KUKA KRL program: EPS_2_25694_AR02_A_20260223033033.src

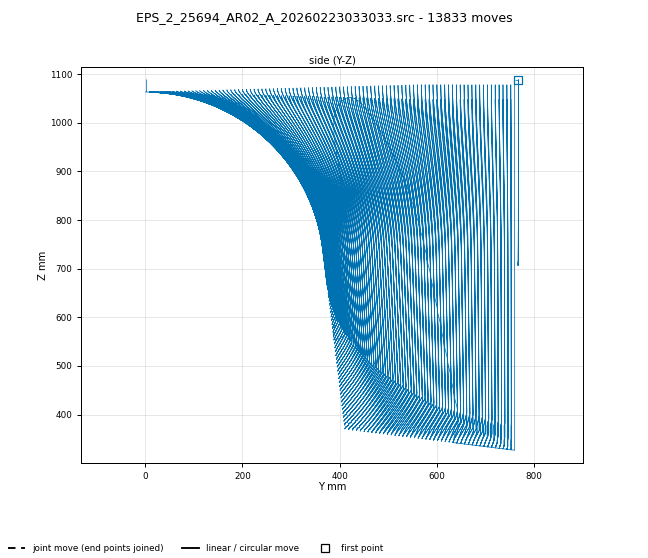
[picture p0: tool path of EPS_2_25694_AR02_A_20260223033033.src, 13833 of 13835 moves have a stored position in this frame; points joined in program order, loops and branches not executed]
&ACCESS RVP
&REL 4
&COMMENT QRS 19112012
&PARAM EDITMASK = *
DEF PART()
EXT BAS (BAS_COMMAND :IN,REAL :IN )
INT I
BAS (#INITMOV,0 )

;KUKA QRS Post kuka4.cps  Date:22-06-2017 !

File_ID=3049

QRS_PRE_INIT()

;Init var - Until changes are made in qrs_pre_init
Outlet_Square_prg=0
Inlet_1_Square_prg=0
Inlet_2_Square_prg=0
Inlet_3_Square_prg=0
Inlet_4_Square_prg=0
Inlet_5_Square_prg=0

Outlet_1={X 0.000, Y 562.000, Z 735.500, B 0.000, E1 0.000 }
Inlet_1={X 0.000, Y 562.000, Z 705.500, B 0.000, E1 180.000 }
Outlet_1_type=686
Inlet_1_type=686
;QRS#1=Sidecore dimensions
;QRS#2=675-27" Concrete
;QRS#3=675-27" Concrete
;QRS#4=
;QRS#5=
;QRS#6=
;QRS#7=
;QRS#8=
;QRS#9=S306-38L
;QRS#10=S306-38L
;QRS#11=
;QRS#12=
;QRS#13=
;QRS#14=
;QRS#15=
;QRS#16=1524x152x1524 5'
;QRS#17=EPS Height
;QRS#18=1078,5
;QRS#19=*
;QRS#20= UPDATED VERSION 22-06-2017
;QRS#21=*
Outlet_Square=0550
Inlet_1_Square=0550
Inlet_2_Square=0
Inlet_3_Square=0
Inlet_4_Square=0
Inlet_5_Square=0
Mill_Square=1
Outlet_Square_Prg=265
Inlet_1_Square_prg=265

QRS_INIT()

$ADVANCE=5

; T1
PTP {E1 173.041,E2 173.041}
PTP {X 0,Y 767.71,A -85,B 0,C 180,E1 173.041,E2 173.041,E3 0,E4 0,E5 0,E6 0}
QRS_SPEED_INIT()
LIN {X 0,Y 767.71,Z 1088.5,A -85,B 0,C 180,E1 173.041,E2 173.041,E3 0,E4 0,E5 0,E6 0} C_VEL
LIN {X 0,Y 767.71,Z 709.31,A -85,B 0,C 180,E1 173.041,E2 173.041} C_VEL
LIN {X 0,Y 767.737,Z 707.31,A -85,B 0,C 180,E1 173.19,E2 173.19} C_VEL
LIN {X 0,Y 767.796,Z 707.31,A -85,B 0,C 180,E1 173.458,E2 173.458} C_VEL
LIN {X 0,Y 767.812,Z 707.31,A -85,B 0,C 180,E1 177.201,E2 177.201} C_VEL
LIN {X 0,Y 767.839,Z 707.31,A -85,B 0,C 180,E1 180.933,E2 180.933} C_VEL
LIN {X 0,Y 767.833,Z 707.31,A -85,B 0,C 180,E1 184.668,E2 184.668} C_VEL
LIN {X 0,Y 767.857,Z 707.31,A -85,B 0,C 180,E1 188.423,E2 188.423} C_VEL
LIN {X 0,Y 767.829,Z 707.31,A -85,B 0,C 180,E1 192.215,E2 192.215} C_VEL
LIN {X 0,Y 767.83,Z 707.31,A -85,B 0,C 180,E1 196.204,E2 196.204} C_VEL
LIN {X 0,Y 767.77,Z 707.31,A -85,B 0,C 180,E1 199.988,E2 199.988} C_VEL
LIN {X 0,Y 767.749,Z 707.31,A -85,B 0,C 180,E1 204.013,E2 204.013} C_VEL
LIN {X 0,Y 767.75,Z 707.31,A -85,B 0,C 180,E1 208.167,E2 208.167} C_VEL
LIN {X 0,Y 767.324,Z 707.31,A -85,B 0,C 180,E1 210.324,E2 210.324} C_VEL
LIN {X 0,Y 767.754,Z 707.31,A -85,B 0,C 180,E1 212.49,E2 212.49} C_VEL
LIN {X 0,Y 767.43,Z 707.31,A -85,B 0,C 180,E1 213.85,E2 213.85} C_VEL
LIN {X 0,Y 767.706,Z 707.31,A -85,B 0,C 180,E1 217.094,E2 217.094} C_VEL
LIN {X 0,Y 767.088,Z 707.31,A -85,B 0,C 180,E1 220.03,E2 220.03} C_VEL
LIN {X 0,Y 767.533,Z 707.31,A -85,B 0,C 180,E1 221.88,E2 221.88} C_VEL
LIN {X 0,Y 767.581,Z 707.31,A -85,B 0,C 180,E1 222.891,E2 222.891} C_VEL
LIN {X 0,Y 767.581,Z 707.31,A -85,B 0,C 180,E1 227.109,E2 227.109} C_VEL
LIN {X 0,Y 767.53,Z 707.31,A -85,B 0,C 180,E1 228.12,E2 228.12} C_VEL
LIN {X 0,Y 767.102,Z 707.31,A -85,B 0,C 180,E1 230.553,E2 230.553} C_VEL
LIN {X 0,Y 767.692,Z 707.31,A -85,B 0,C 180,E1 232.964,E2 232.964} C_VEL
LIN {X 0,Y 767.598,Z 707.31,A -85,B 0,C 180,E1 236.132,E2 236.132} C_VEL
LIN {X 0,Y 767.614,Z 707.31,A -85,B 0,C 180,E1 237.503,E2 237.503} C_VEL
LIN {X 0,Y 767.641,Z 707.31,A -85,B 0,C 180,E1 239.69,E2 239.69} C_VEL
LIN {X 0,Y 767.411,Z 728.971,A -85,B 0,C 180,E1 240.873,E2 240.873} C_VEL
LIN {X 0,Y 767.537,Z 761.793,A -85,B 0,C 180,E1 241.233,E2 241.233} C_VEL
LIN {X 0,Y 767.433,Z 775.286,A -85,B 0,C 180,E1 241.406,E2 241.406} C_VEL
LIN {X 0,Y 767.548,Z 791.123,A -85,B 0,C 180,E1 241.677,E2 241.677} C_VEL
LIN {X 0,Y 767.449,Z 807.75,A -85,B 0,C 180,E1 242.019,E2 242.019} C_VEL
LIN {X 0,Y 767.663,Z 824.864,A -85,B 0,C 180,E1 242.456,E2 242.456} C_VEL
LIN {X 0,Y 767.66,Z 840.823,A -85,B 0,C 180,E1 242.921,E2 242.921} C_VEL
LIN {X 0,Y 767.553,Z 854.893,A -85,B 0,C 180,E1 243.38,E2 243.38} C_VEL
LIN {X 0,Y 767.694,Z 871.263,A -85,B 0,C 180,E1 243.998,E2 243.998} C_VEL
LIN {X 0,Y 767.655,Z 888.029,A -85,B 0,C 180,E1 244.706,E2 244.706} C_VEL
LIN {X 0,Y 767.705,Z 901.802,A -85,B 0,C 180,E1 245.351,E2 245.351} C_VEL
LIN {X 0,Y 767.712,Z 916.578,A -85,B 0,C 180,E1 246.114,E2 246.114} C_VEL
LIN {X 0,Y 767.693,Z 930.073,A -85,B 0,C 180,E1 246.876,E2 246.876} C_VEL
LIN {X 0,Y 767.691,Z 942.43,A -85,B 0,C 180,E1 247.634,E2 247.634} C_VEL
LIN {X 0,Y 767.701,Z 955.671,A -85,B 0,C 180,E1 248.523,E2 248.523} C_VEL
LIN {X 0,Y 767.718,Z 968.193,A -85,B 0,C 180,E1 249.439,E2 249.439} C_VEL
LIN {X 0,Y 767.619,Z 980.057,A -85,B 0,C 180,E1 250.38,E2 250.38} C_VEL
LIN {X 0,Y 767.656,Z 990.133,A -85,B 0,C 180,E1 251.245,E2 251.245} C_VEL
LIN {X 0,Y 767.778,Z 1000.684,A -85,B 0,C 180,E1 252.23,E2 252.23} C_VEL
LIN {X 0,Y 767.637,Z 1011.458,A -85,B 0,C 180,E1 253.326,E2 253.326} C_VEL
LIN {X 0,Y 767.699,Z 1020.42,A -85,B 0,C 180,E1 254.322,E2 254.322} C_VEL
LIN {X 0,Y 767.767,Z 1028.417,A -85,B 0,C 180,E1 255.29,E2 255.29} C_VEL
LIN {X 0,Y 767.624,Z 1037.823,A -85,B 0,C 180,E1 256.546,E2 256.546} C_VEL
LIN {X 0,Y 767.75,Z 1044.548,A -85,B 0,C 180,E1 257.545,E2 257.545} C_VEL
LIN {X 0,Y 767.749,Z 1048.907,A -85,B 0,C 180,E1 258.26,E2 258.26} C_VEL
LIN {X 0,Y 767.595,Z 1053.115,A -85,B 0,C 180,E1 258.971,E2 258.971} C_VEL
LIN {X 0,Y 767.579,Z 1059.347,A -85,B 0,C 180,E1 260.157,E2 260.157} C_VEL
LIN {X 0,Y 767.814,Z 1064.751,A -85,B 0,C 180,E1 261.341,E2 261.341} C_VEL
LIN {X 0,Y 767.552,Z 1069.482,A -85,B 0,C 180,E1 262.516,E2 262.516} C_VEL
LIN {X 0,Y 767.638,Z 1073.816,A -85,B 0,C 180,E1 263.832,E2 263.832} C_VEL
LIN {X 0,Y 767.832,Z 1075.821,A -85,B 0,C 180,E1 264.583,E2 264.583} C_VEL
LIN {X 0,Y 767.656,Z 1077.679,A -85,B 0,C 180,E1 265.331,E2 265.331} C_VEL
LIN {X 0,Y 767.552,Z 1079.276,A -85,B 0,C 180,E1 266.079,E2 266.079} C_VEL
LIN {X 0,Y 767.665,Z 1081.027,A -85,B 0,C 180,E1 267.201,E2 267.201} C_VEL
LIN {X 0,Y 767.713,Z 1082.196,A -85,B 0,C 180,E1 268.321,E2 268.321} C_VEL
LIN {X 0,Y 767.556,Z 1082.708,A -85,B 0,C 180,E1 269.067,E2 269.067} C_VEL
LIN {X 0,Y 767.7,Z 1082.68,A -85,B 0,C 180,E1 270.933,E2 270.933} C_VEL
LIN {X 0,Y 767.651,Z 1081.876,A -85,B 0,C 180,E1 272.052,E2 272.052} C_VEL
LIN {X 0,Y 767.525,Z 1081.053,A -85,B 0,C 180,E1 272.8,E2 272.8} C_VEL
LIN {X 0,Y 767.569,Z 1079.273,A -85,B 0,C 180,E1 273.921,E2 273.921} C_VEL
LIN {X 0,Y 767.76,Z 1077.66,A -85,B 0,C 180,E1 274.668,E2 274.668} C_VEL
LIN {X 0,Y 767.653,Z 1074.831,A -85,B 0,C 180,E1 275.793,E2 275.793} C_VEL
LIN {X 0,Y 767.602,Z 1072.628,A -85,B 0,C 180,E1 276.544,E2 276.544} C_VEL
LIN {X 0,Y 767.713,Z 1069.455,A -85,B 0,C 180,E1 277.483,E2 277.483} C_VEL
LIN {X 0,Y 767.824,Z 1067.577,A -85,B 0,C 180,E1 277.952,E2 277.952} C_VEL
LIN {X 0,Y 767.62,Z 1063.757,A -85,B 0,C 180,E1 278.897,E2 278.897} C_VEL
LIN {X 0,Y 767.559,Z 1058.195,A -85,B 0,C 180,E1 280.08,E2 280.08} C_VEL
LIN {X 0,Y 767.835,Z 1051.779,A -85,B 0,C 180,E1 281.263,E2 281.263} C_VEL
LIN {X 0,Y 767.624,Z 1044.562,A -85,B 0,C 180,E1 282.457,E2 282.457} C_VEL
LIN {X 0,Y 767.658,Z 1036.703,A -85,B 0,C 180,E1 283.612,E2 283.612} C_VEL
LIN {X 0,Y 767.821,Z 1029.879,A -85,B 0,C 180,E1 284.516,E2 284.516} C_VEL
LIN {X 0,Y 767.629,Z 1020.425,A -85,B 0,C 180,E1 285.679,E2 285.679} C_VEL
LIN {X 0,Y 767.731,Z 1009.176,A -85,B 0,C 180,E1 286.916,E2 286.916} C_VEL
LIN {X 0,Y 767.752,Z 999.435,A -85,B 0,C 180,E1 287.893,E2 287.893} C_VEL
LIN {X 0,Y 767.658,Z 988.765,A -85,B 0,C 180,E1 288.878,E2 288.878} C_VEL
LIN {X 0,Y 767.742,Z 977.061,A -85,B 0,C 180,E1 289.864,E2 289.864} C_VEL
LIN {X 0,Y 767.717,Z 964.937,A -85,B 0,C 180,E1 290.806,E2 290.806} C_VEL
LIN {X 0,Y 767.695,Z 954,A -85,B 0,C 180,E1 291.594,E2 291.594} C_VEL
LIN {X 0,Y 767.712,Z 940.408,A -85,B 0,C 180,E1 292.491,E2 292.491} C_VEL
LIN {X 0,Y 767.708,Z 926.801,A -85,B 0,C 180,E1 293.314,E2 293.314} C_VEL
LIN {X 0,Y 767.702,Z 913.126,A -85,B 0,C 180,E1 294.071,E2 294.071} C_VEL
LIN {X 0,Y 767.609,Z 898.313,A -85,B 0,C 180,E1 294.82,E2 294.82} C_VEL
LIN {X 0,Y 767.699,Z 884.655,A -85,B 0,C 180,E1 295.444,E2 295.444} C_VEL
LIN {X 0,Y 767.675,Z 869.453,A -85,B 0,C 180,E1 296.074,E2 296.074} C_VEL
LIN {X 0,Y 767.622,Z 855.717,A -85,B 0,C 180,E1 296.587,E2 296.587} C_VEL
LIN {X 0,Y 767.679,Z 837.479,A -85,B 0,C 180,E1 297.183,E2 297.183} C_VEL
LIN {X 0,Y 767.517,Z 820.548,A -85,B 0,C 180,E1 297.665,E2 297.665} C_VEL
LIN {X 0,Y 767.57,Z 810.447,A -85,B 0,C 180,E1 297.91,E2 297.91} C_VEL
LIN {X 0,Y 767.621,Z 801.598,A -85,B 0,C 180,E1 298.106,E2 298.106} C_VEL
LIN {X 0,Y 767.599,Z 787.941,A -85,B 0,C 180,E1 298.38,E2 298.38} C_VEL
LIN {X 0,Y 767.429,Z 775.322,A -85,B 0,C 180,E1 298.593,E2 298.593} C_VEL
LIN {X 0,Y 767.549,Z 757.094,A -85,B 0,C 180,E1 298.825,E2 298.825} C_VEL
LIN {X 0,Y 767.411,Z 729.395,A -85,B 0,C 180,E1 299.122,E2 299.122} C_VEL
LIN {X 0,Y 767.689,Z 707.31,A -85,B 0,C 180,E1 300.308,E2 300.308} C_VEL
LIN {X 0,Y 767.796,Z 707.31,A -85,B 0,C 180,E1 302.488,E2 302.488} C_VEL
LIN {X 0,Y 767.259,Z 707.31,A -85,B 0,C 180,E1 304.756,E2 304.756} C_VEL
LIN {X 0,Y 767.698,Z 707.31,A -85,B 0,C 180,E1 307.093,E2 307.093} C_VEL
LIN {X 0,Y 767.134,Z 707.31,A -85,B 0,C 180,E1 310.034,E2 310.034} C_VEL
LIN {X 0,Y 767.63,Z 707.31,A -85,B 0,C 180,E1 311.873,E2 311.873} C_VEL
LIN {X 0,Y 767.669,Z 707.31,A -85,B 0,C 180,E1 312.898,E2 312.898} C_VEL
LIN {X 0,Y 767.67,Z 707.31,A -85,B 0,C 180,E1 314.427,E2 314.427} C_VEL
LIN {X 0,Y 767.632,Z 707.31,A -85,B 0,C 180,E1 315.57,E2 315.57} C_VEL
LIN {X 0,Y 767.641,Z 707.31,A -85,B 0,C 180,E1 319.92,E2 319.92} C_VEL
LIN {X 0,Y 767.641,Z 707.31,A -85,B 0,C 180,E1 320.586,E2 320.586} C_VEL
LIN {X 0,Y 767.199,Z 707.31,A -85,B 0,C 180,E1 322.956,E2 322.956} C_VEL
LIN {X 0,Y 767.714,Z 707.31,A -85,B 0,C 180,E1 325.268,E2 325.268} C_VEL
LIN {X 0,Y 767.766,Z 707.31,A -85,B 0,C 180,E1 329.62,E2 329.62} C_VEL
LIN {X 0,Y 767.768,Z 707.31,A -85,B 0,C 180,E1 333.539,E2 333.539} C_VEL
LIN {X 0,Y 767.758,Z 707.31,A -85,B 0,C 180,E1 333.929,E2 333.929} C_VEL
LIN {X 0,Y 767.757,Z 707.31,A -85,B 0,C 180,E1 338.014,E2 338.014} C_VEL
LIN {X 0,Y 767.788,Z 707.31,A -85,B 0,C 180,E1 341.985,E2 341.985} C_VEL
LIN {X 0,Y 767.515,Z 707.31,A -85,B 0,C 180,E1 343.931,E2 343.931} C_VEL
LIN {X 0,Y 767.673,Z 707.31,A -85,B 0,C 180,E1 345.866,E2 345.866} C_VEL
LIN {X 0,Y 767.85,Z 707.31,A -85,B 0,C 180,E1 349.687,E2 349.687} C_VEL
LIN {X 0,Y 767.871,Z 707.31,A -85,B 0,C 180,E1 353.458,E2 353.458} C_VEL
LIN {X 0,Y 767.844,Z 707.31,A -85,B 0,C 180,E1 357.201,E2 357.201} C_VEL
LIN {X 0,Y 767.813,Z 707.31,A -85,B 0,C 180,E1 360.933,E2 360.933} C_VEL
LIN {X 0,Y 767.806,Z 707.31,A -85,B 0,C 180,E1 364.668,E2 364.668} C_VEL
LIN {X 0,Y 767.794,Z 707.31,A -85,B 0,C 180,E1 368.424,E2 368.424} C_VEL
LIN {X 0,Y 767.808,Z 707.31,A -85,B 0,C 180,E1 372.216,E2 372.216} C_VEL
LIN {X 0,Y 767.849,Z 707.31,A -85,B 0,C 180,E1 376.209,E2 376.209} C_VEL
LIN {X 0,Y 767.798,Z 707.31,A -85,B 0,C 180,E1 379.987,E2 379.987} C_VEL
LIN {X 0,Y 767.788,Z 707.31,A -85,B 0,C 180,E1 384.011,E2 384.011} C_VEL
LIN {X 0,Y 767.772,Z 707.31,A -85,B 0,C 180,E1 388.166,E2 388.166} C_VEL
LIN {X 0,Y 767.323,Z 707.31,A -85,B 0,C 180,E1 390.324,E2 390.324} C_VEL
LIN {X 0,Y 767.706,Z 707.31,A -85,B 0,C 180,E1 392.493,E2 392.493} C_VEL
LIN {X 0,Y 767.384,Z 707.31,A -85,B 0,C 180,E1 393.845,E2 393.845} C_VEL
LIN {X 0,Y 767.666,Z 707.31,A -85,B 0,C 180,E1 397.09,E2 397.09} C_VEL
LIN {X 0,Y 767.085,Z 707.31,A -85,B 0,C 180,E1 400.03,E2 400.03} C_VEL
LIN {X 0,Y 767.568,Z 707.31,A -85,B 0,C 180,E1 401.877,E2 401.877} C_VEL
LIN {X 0,Y 767.619,Z 707.31,A -85,B 0,C 180,E1 402.894,E2 402.894} C_VEL
LIN {X 0,Y 767.576,Z 707.31,A -85,B 0,C 180,E1 407.109,E2 407.109} C_VEL
LIN {X 0,Y 767.531,Z 707.31,A -85,B 0,C 180,E1 408.12,E2 408.12} C_VEL
LIN {X 0,Y 767.121,Z 707.31,A -85,B 0,C 180,E1 410.555,E2 410.555} C_VEL
LIN {X 0,Y 767.734,Z 707.31,A -85,B 0,C 180,E1 412.967,E2 412.967} C_VEL
LIN {X 0,Y 767.634,Z 707.31,A -85,B 0,C 180,E1 416.127,E2 416.127} C_VEL
LIN {X 0,Y 767.601,Z 707.31,A -85,B 0,C 180,E1 417.503,E2 417.503} C_VEL
LIN {X 0,Y 767.858,Z 707.31,A -85,B 0,C 180,E1 420.635,E2 420.635} C_VEL
LIN {X 0,Y 766.716,Z 707.31,A -85,B 0,C 180,E1 420.886,E2 420.886} C_VEL
LIN {X 0,Y 767.333,Z 731.466,A -85,B 0,C 180,E1 421.176,E2 421.176} C_VEL
LIN {X 0,Y 767.435,Z 745.357,A -85,B 0,C 180,E1 421.363,E2 421.363} C_VEL
LIN {X 0,Y 767.54,Z 761.823,A -85,B 0,C 180,E1 421.646,E2 421.646} C_VEL
LIN {X 0,Y 767.454,Z 778.242,A -85,B 0,C 180,E1 421.986,E2 421.986} C_VEL
LIN {X 0,Y 767.631,Z 794.143,A -85,B 0,C 180,E1 422.389,E2 422.389} C_VEL
LIN {X 0,Y 767.586,Z 811.017,A -85,B 0,C 180,E1 422.879,E2 422.879} C_VEL
LIN {X 0,Y 767.597,Z 821.633,A -85,B 0,C 180,E1 423.229,E2 423.229} C_VEL
LIN {X 0,Y 767.652,Z 830.77,A -85,B 0,C 180,E1 423.557,E2 423.557} C_VEL
LIN {X 0,Y 767.67,Z 842.534,A -85,B 0,C 180,E1 424.005,E2 424.005} C_VEL
LIN {X 0,Y 767.616,Z 857.298,A -85,B 0,C 180,E1 424.625,E2 424.625} C_VEL
LIN {X 0,Y 767.704,Z 872.822,A -85,B 0,C 180,E1 425.358,E2 425.358} C_VEL
LIN {X 0,Y 767.706,Z 886.246,A -85,B 0,C 180,E1 426.05,E2 426.05} C_VEL
LIN {X 0,Y 767.699,Z 900.808,A -85,B 0,C 180,E1 426.876,E2 426.876} C_VEL
LIN {X 0,Y 767.715,Z 913.106,A -85,B 0,C 180,E1 427.635,E2 427.635} C_VEL
LIN {X 0,Y 767.732,Z 926.109,A -85,B 0,C 180,E1 428.51,E2 428.51} C_VEL
LIN {X 0,Y 767.692,Z 937.694,A -85,B 0,C 180,E1 429.354,E2 429.354} C_VEL
LIN {X 0,Y 767.693,Z 949.134,A -85,B 0,C 180,E1 430.258,E2 430.258} C_VEL
LIN {X 0,Y 767.755,Z 960.62,A -85,B 0,C 180,E1 431.248,E2 431.248} C_VEL
LIN {X 0,Y 767.617,Z 971.133,A -85,B 0,C 180,E1 432.226,E2 432.226} C_VEL
LIN {X 0,Y 767.635,Z 980.763,A -85,B 0,C 180,E1 433.204,E2 433.204} C_VEL
LIN {X 0,Y 767.794,Z 990.787,A -85,B 0,C 180,E1 434.324,E2 434.324} C_VEL
LIN {X 0,Y 767.595,Z 998.788,A -85,B 0,C 180,E1 435.287,E2 435.287} C_VEL
LIN {X 0,Y 767.635,Z 1008.181,A -85,B 0,C 180,E1 436.555,E2 436.555} C_VEL
LIN {X 0,Y 767.838,Z 1014.839,A -85,B 0,C 180,E1 437.546,E2 437.546} C_VEL
LIN {X 0,Y 767.606,Z 1022.075,A -85,B 0,C 180,E1 438.734,E2 438.734} C_VEL
LIN {X 0,Y 767.688,Z 1028.418,A -85,B 0,C 180,E1 439.922,E2 439.922} C_VEL
LIN {X 0,Y 767.815,Z 1031.726,A -85,B 0,C 180,E1 440.633,E2 440.633} C_VEL
LIN {X 0,Y 767.696,Z 1033.956,A -85,B 0,C 180,E1 441.104,E2 441.104} C_VEL
LIN {X 0,Y 767.567,Z 1039.63,A -85,B 0,C 180,E1 442.516,E2 442.516} C_VEL
LIN {X 0,Y 767.836,Z 1043.902,A -85,B 0,C 180,E1 443.833,E2 443.833} C_VEL
LIN {X 0,Y 767.651,Z 1045.978,A -85,B 0,C 180,E1 444.582,E2 444.582} C_VEL
LIN {X 0,Y 767.527,Z 1047.797,A -85,B 0,C 180,E1 445.33,E2 445.33} C_VEL
LIN {X 0,Y 767.528,Z 1049.376,A -85,B 0,C 180,E1 446.079,E2 446.079} C_VEL
LIN {X 0,Y 767.766,Z 1051.076,A -85,B 0,C 180,E1 447.201,E2 447.201} C_VEL
LIN {X 0,Y 767.683,Z 1051.909,A -85,B 0,C 180,E1 447.948,E2 447.948} C_VEL
LIN {X 0,Y 767.503,Z 1052.73,A -85,B 0,C 180,E1 449.067,E2 449.067} C_VEL
LIN {X 0,Y 767.839,Z 1052.64,A -85,B 0,C 180,E1 450.933,E2 450.933} C_VEL
LIN {X 0,Y 767.651,Z 1052.167,A -85,B 0,C 180,E1 451.679,E2 451.679} C_VEL
LIN {X 0,Y 767.568,Z 1050.977,A -85,B 0,C 180,E1 452.8,E2 452.8} C_VEL
LIN {X 0,Y 767.769,Z 1049.14,A -85,B 0,C 180,E1 453.92,E2 453.92} C_VEL
LIN {X 0,Y 767.722,Z 1047.573,A -85,B 0,C 180,E1 454.669,E2 454.669} C_VEL
LIN {X 0,Y 767.556,Z 1044.725,A -85,B 0,C 180,E1 455.794,E2 455.794} C_VEL
LIN {X 0,Y 767.553,Z 1043.709,A -85,B 0,C 180,E1 456.169,E2 456.169} C_VEL
LIN {X 0,Y 767.803,Z 1039.283,A -85,B 0,C 180,E1 457.482,E2 457.482} C_VEL
LIN {X 0,Y 767.581,Z 1033.551,A -85,B 0,C 180,E1 458.898,E2 458.898} C_VEL
LIN {X 0,Y 767.696,Z 1027.934,A -85,B 0,C 180,E1 460.078,E2 460.078} C_VEL
LIN {X 0,Y 767.795,Z 1024.114,A -85,B 0,C 180,E1 460.788,E2 460.788} C_VEL
LIN {X 0,Y 767.632,Z 1020.089,A -85,B 0,C 180,E1 461.504,E2 461.504} C_VEL
LIN {X 0,Y 767.584,Z 1014.26,A -85,B 0,C 180,E1 462.458,E2 462.458} C_VEL
LIN {X 0,Y 767.802,Z 1006.2,A -85,B 0,C 180,E1 463.63,E2 463.63} C_VEL
LIN {X 0,Y 767.611,Z 998.056,A -85,B 0,C 180,E1 464.713,E2 464.713} C_VEL
LIN {X 0,Y 767.603,Z 988.335,A -85,B 0,C 180,E1 465.874,E2 465.874} C_VEL
LIN {X 0,Y 767.79,Z 978.725,A -85,B 0,C 180,E1 466.915,E2 466.915} C_VEL
LIN {X 0,Y 767.663,Z 968.946,A -85,B 0,C 180,E1 467.895,E2 467.895} C_VEL
LIN {X 0,Y 767.674,Z 958.234,A -85,B 0,C 180,E1 468.878,E2 468.878} C_VEL
LIN {X 0,Y 767.733,Z 946.486,A -85,B 0,C 180,E1 469.865,E2 469.865} C_VEL
LIN {X 0,Y 767.676,Z 936.03,A -85,B 0,C 180,E1 470.683,E2 470.683} C_VEL
LIN {X 0,Y 767.702,Z 923.158,A -85,B 0,C 180,E1 471.605,E2 471.605} C_VEL
LIN {X 0,Y 767.72,Z 909.669,A -85,B 0,C 180,E1 472.491,E2 472.491} C_VEL
LIN {X 0,Y 767.698,Z 897.13,A -85,B 0,C 180,E1 473.251,E2 473.251} C_VEL
LIN {X 0,Y 767.661,Z 883.363,A -85,B 0,C 180,E1 474.016,E2 474.016} C_VEL
LIN {X 0,Y 767.709,Z 868.143,A -85,B 0,C 180,E1 474.779,E2 474.779} C_VEL
LIN {X 0,Y 767.676,Z 854.017,A -85,B 0,C 180,E1 475.427,E2 475.427} C_VEL
LIN {X 0,Y 767.64,Z 840.173,A -85,B 0,C 180,E1 476.003,E2 476.003} C_VEL
LIN {X 0,Y 767.674,Z 822.353,A -85,B 0,C 180,E1 476.655,E2 476.655} C_VEL
LIN {X 0,Y 767.539,Z 807.048,A -85,B 0,C 180,E1 477.155,E2 477.155} C_VEL
LIN {X 0,Y 767.67,Z 790.049,A -85,B 0,C 180,E1 477.626,E2 477.626} C_VEL
LIN {X 0,Y 767.643,Z 774.248,A -85,B 0,C 180,E1 478.006,E2 478.006} C_VEL
LIN {X 0,Y 767.488,Z 760.439,A -85,B 0,C 180,E1 478.294,E2 478.294} C_VEL
LIN {X 0,Y 767.647,Z 741.352,A -85,B 0,C 180,E1 478.599,E2 478.599} C_VEL
LIN {X 0,Y 767.413,Z 720.586,A -85,B 0,C 180,E1 478.855,E2 478.855} C_VEL
LIN {X 0,Y 767.103,Z 715.733,A -85,B 0,C 180,E1 478.919,E2 478.919} C_VEL
LIN {X 0,Y 765.967,Z 707.31,A -85,B 0,C 180,E1 479.059,E2 479.059} C_VEL
LIN {X 0,Y 767.879,Z 707.31,A -85,B 0,C 180,E1 479.317,E2 479.317} C_VEL
LIN {X 0,Y 767.752,Z 707.31,A -85,B 0,C 180,E1 482.49,E2 482.49} C_VEL
LIN {X 0,Y 767.418,Z 707.31,A -85,B 0,C 180,E1 483.848,E2 483.848} C_VEL
LIN {X 0,Y 767.742,Z 707.31,A -85,B 0,C 180,E1 487.098,E2 487.098} C_VEL
LIN {X 0,Y 767.157,Z 707.31,A -85,B 0,C 180,E1 490.036,E2 490.036} C_VEL
LIN {X 0,Y 767.638,Z 707.31,A -85,B 0,C 180,E1 491.873,E2 491.873} C_VEL
LIN {X 0,Y 767.66,Z 707.31,A -85,B 0,C 180,E1 492.897,E2 492.897} C_VEL
LIN {X 0,Y 767.674,Z 707.31,A -85,B 0,C 180,E1 494.427,E2 494.427} C_VEL
LIN {X 0,Y 767.645,Z 707.31,A -85,B 0,C 180,E1 495.571,E2 495.571} C_VEL
LIN {X 0,Y 767.662,Z 707.31,A -85,B 0,C 180,E1 499.919,E2 499.919} C_VEL
LIN {X 0,Y 767.649,Z 707.31,A -85,B 0,C 180,E1 500.587,E2 500.587} C_VEL
LIN {X 0,Y 767.201,Z 707.31,A -85,B 0,C 180,E1 502.956,E2 502.956} C_VEL
LIN {X 0,Y 767.688,Z 707.31,A -85,B 0,C 180,E1 505.267,E2 505.267} C_VEL
LIN {X 0,Y 767.773,Z 707.31,A -85,B 0,C 180,E1 509.619,E2 509.619} C_VEL
LIN {X 0,Y 767.792,Z 707.31,A -85,B 0,C 180,E1 513.536,E2 513.536} C_VEL
LIN {X 0,Y 767.79,Z 707.31,A -85,B 0,C 180,E1 513.93,E2 513.93} C_VEL
LIN {X 0,Y 767.81,Z 707.31,A -85,B 0,C 180,E1 518.016,E2 518.016} C_VEL
LIN {X 0,Y 767.831,Z 707.31,A -85,B 0,C 180,E1 521.987,E2 521.987} C_VEL
LIN {X 0,Y 767.502,Z 707.31,A -85,B 0,C 180,E1 523.93,E2 523.93} C_VEL
LIN {X 0,Y 767.619,Z 707.31,A -85,B 0,C 180,E1 525.865,E2 525.865} C_VEL
LIN {X 0,Y 767.814,Z 707.31,A -85,B 0,C 180,E1 529.686,E2 529.686} C_VEL
LIN {X 0,Y 767.737,Z 707.31,A -85,B 0,C 180,E1 533.19,E2 533.19} C_VEL
LIN {X 0,Y 767.797,Z 709.31,A -85,B 0,C 180,E1 533.34,E2 533.34} C_VEL
LIN {X 0,Y 767.797,Z 1088.5,A -85,B 0,C 180,E1 533.34,E2 533.34} C_VEL
LIN {X 0,Y 767.797,Z 1088.5,A -85,B 0,C 180,E1 533.34,E2 533.34}

QRS_NEXT_CUT()
PTP {E1 537.316,E2 537.316}
PTP {X 0,Y 759.845,A -85,B 0,C 180,E1 537.316,E2 537.316,E3 0,E4 0,E5 0,E6 0}
QRS_SPEED_INIT()
LIN {X 0,Y 759.845,Z 1088.5,A -85,B 0,C 180,E1 537.316,E2 537.316,E3 0,E4 0,E5 0,E6 0} C_VEL
LIN {X 0,Y 759.845,Z 336.65,A -85,B 0,C 180,E1 537.316,E2 537.316} C_VEL
LIN {X 0,Y 759.845,Z 328.572,A -85,B 0,C 180,E1 537.316,E2 537.316} C_VEL
LIN {X 0,Y 759.845,Z 326.572,A -85,B 0,C 180,E1 537.165,E2 537.165} C_VEL
LIN {X 0,Y 759.903,Z 326.568,A -85,B 0,C 180,E1 534.488,E2 534.488} C_VEL
LIN {X 0,Y 759.869,Z 326.575,A -85,B 0,C 180,E1 531.601,E2 531.601} C_VEL
LIN {X 0,Y 759.845,Z 326.572,A -85,B 0,C 180,E1 529.077,E2 529.077} C_VEL
LIN {X 0,Y 759.89,Z 326.569,A -85,B 0,C 180,E1 526.454,E2 526.454} C_VEL
LIN {X 0,Y 759.873,Z 326.575,A -85,B 0,C 180,E1 523.487,E2 523.487} C_VEL
LIN {X 0,Y 759.846,Z 326.572,A -85,B 0,C 180,E1 520.953,E2 520.953} C_VEL
LIN {X 0,Y 759.881,Z 326.569,A -85,B 0,C 180,E1 518.381,E2 518.381} C_VEL
LIN {X 0,Y 759.873,Z 326.575,A -85,B 0,C 180,E1 515.346,E2 515.346} C_VEL
LIN {X 0,Y 759.847,Z 326.572,A -85,B 0,C 180,E1 512.817,E2 512.817} C_VEL
LIN {X 0,Y 759.891,Z 326.568,A -85,B 0,C 180,E1 510.173,E2 510.173} C_VEL
LIN {X 0,Y 759.87,Z 326.575,A -85,B 0,C 180,E1 507.17,E2 507.17} C_VEL
LIN {X 0,Y 759.848,Z 326.572,A -85,B 0,C 180,E1 504.62,E2 504.62} C_VEL
LIN {X 0,Y 759.899,Z 326.568,A -85,B 0,C 180,E1 501.989,E2 501.989} C_VEL
LIN {X 0,Y 759.873,Z 326.575,A -85,B 0,C 180,E1 499.052,E2 499.052} C_VEL
LIN {X 0,Y 759.849,Z 326.572,A -85,B 0,C 180,E1 496.474,E2 496.474} C_VEL
LIN {X 0,Y 759.916,Z 326.567,A -85,B 0,C 180,E1 493.749,E2 493.749} C_VEL
LIN {X 0,Y 759.866,Z 326.575,A -85,B 0,C 180,E1 490.832,E2 490.832} C_VEL
LIN {X 0,Y 759.85,Z 326.572,A -85,B 0,C 180,E1 488.301,E2 488.301} C_VEL
LIN {X 0,Y 759.911,Z 326.569,A -85,B 0,C 180,E1 485.593,E2 485.593} C_VEL
LIN {X 0,Y 759.85,Z 326.665,A -85,B 0,C 180,E1 484.249,E2 484.249} C_VEL
LIN {X 0,Y 759.884,Z 347.573,A -85,B 0,C 180,E1 482.756,E2 482.756} C_VEL
LIN {X 0,Y 759.914,Z 586.155,A -85,B 0,C 180,E1 480.163,E2 480.163} C_VEL
LIN {X 0,Y 759.918,Z 735.836,A -85,B 0,C 180,E1 478.552,E2 478.552} C_VEL
LIN {X 0,Y 759.897,Z 759.154,A -85,B 0,C 180,E1 478.189,E2 478.189} C_VEL
LIN {X 0,Y 759.902,Z 781.501,A -85,B 0,C 180,E1 477.701,E2 477.701} C_VEL
LIN {X 0,Y 759.897,Z 801.388,A -85,B 0,C 180,E1 477.167,E2 477.167} C_VEL
LIN {X 0,Y 759.919,Z 824.793,A -85,B 0,C 180,E1 476.406,E2 476.406} C_VEL
LIN {X 0,Y 759.916,Z 845.178,A -85,B 0,C 180,E1 475.61,E2 475.61} C_VEL
LIN {X 0,Y 759.913,Z 864.717,A -85,B 0,C 180,E1 474.735,E2 474.735} C_VEL
LIN {X 0,Y 759.912,Z 886.993,A -85,B 0,C 180,E1 473.578,E2 473.578} C_VEL
LIN {X 0,Y 759.914,Z 904.978,A -85,B 0,C 180,E1 472.513,E2 472.513} C_VEL
LIN {X 0,Y 759.906,Z 925.463,A -85,B 0,C 180,E1 471.133,E2 471.133} C_VEL
LIN {X 0,Y 759.916,Z 942.7,A -85,B 0,C 180,E1 469.815,E2 469.815} C_VEL
LIN {X 0,Y 759.916,Z 959.761,A -85,B 0,C 180,E1 468.329,E2 468.329} C_VEL
LIN {X 0,Y 759.898,Z 975.058,A -85,B 0,C 180,E1 466.827,E2 466.827} C_VEL
LIN {X 0,Y 759.912,Z 989.594,A -85,B 0,C 180,E1 465.179,E2 465.179} C_VEL
LIN {X 0,Y 759.908,Z 1001.089,A -85,B 0,C 180,E1 463.7,E2 463.7} C_VEL
LIN {X 0,Y 759.903,Z 1012.978,A -85,B 0,C 180,E1 461.922,E2 461.922} C_VEL
LIN {X 0,Y 759.908,Z 1021.724,A -85,B 0,C 180,E1 460.385,E2 460.385} C_VEL
LIN {X 0,Y 759.89,Z 1030.202,A -85,B 0,C 180,E1 458.627,E2 458.627} C_VEL
LIN {X 0,Y 759.914,Z 1036.829,A -85,B 0,C 180,E1 456.877,E2 456.877} C_VEL
LIN {X 0,Y 759.901,Z 1041.594,A -85,B 0,C 180,E1 455.285,E2 455.285} C_VEL
LIN {X 0,Y 759.907,Z 1045.717,A -85,B 0,C 180,E1 453.319,E2 453.319} C_VEL
LIN {X 0,Y 759.898,Z 1047.657,A -85,B 0,C 180,E1 451.734,E2 451.734} C_VEL
LIN {X 0,Y 759.911,Z 1048.497,A -85,B 0,C 180,E1 449.925,E2 449.925} C_VEL
LIN {X 0,Y 759.908,Z 1047.603,A -85,B 0,C 180,E1 448.115,E2 448.115} C_VEL
LIN {X 0,Y 759.912,Z 1045.289,A -85,B 0,C 180,E1 446.303,E2 446.303} C_VEL
LIN {X 0,Y 759.893,Z 1041.221,A -85,B 0,C 180,E1 444.488,E2 444.488} C_VEL
LIN {X 0,Y 759.919,Z 1036.368,A -85,B 0,C 180,E1 442.895,E2 442.895} C_VEL
LIN {X 0,Y 759.905,Z 1028.873,A -85,B 0,C 180,E1 440.991,E2 440.991} C_VEL
LIN {X 0,Y 759.899,Z 1020.978,A -85,B 0,C 180,E1 439.385,E2 439.385} C_VEL
LIN {X 0,Y 759.917,Z 1011.204,A -85,B 0,C 180,E1 437.692,E2 437.692} C_VEL
LIN {X 0,Y 759.909,Z 999.442,A -85,B 0,C 180,E1 435.989,E2 435.989} C_VEL
LIN {X 0,Y 759.91,Z 987.765,A -85,B 0,C 180,E1 434.508,E2 434.508} C_VEL
LIN {X 0,Y 759.905,Z 972.836,A -85,B 0,C 180,E1 432.858,E2 432.858} C_VEL
LIN {X 0,Y 759.903,Z 958.171,A -85,B 0,C 180,E1 431.432,E2 431.432} C_VEL
LIN {X 0,Y 759.915,Z 940.414,A -85,B 0,C 180,E1 429.914,E2 429.914} C_VEL
LIN {X 0,Y 759.917,Z 922.823,A -85,B 0,C 180,E1 428.584,E2 428.584} C_VEL
LIN {X 0,Y 759.913,Z 903.788,A -85,B 0,C 180,E1 427.323,E2 427.323} C_VEL
LIN {X 0,Y 759.91,Z 885.673,A -85,B 0,C 180,E1 426.257,E2 426.257} C_VEL
LIN {X 0,Y 759.914,Z 863.082,A -85,B 0,C 180,E1 425.099,E2 425.099} C_VEL
LIN {X 0,Y 759.917,Z 844.331,A -85,B 0,C 180,E1 424.265,E2 424.265} C_VEL
LIN {X 0,Y 759.914,Z 822.667,A -85,B 0,C 180,E1 423.425,E2 423.425} C_VEL
LIN {X 0,Y 759.902,Z 800.83,A -85,B 0,C 180,E1 422.727,E2 422.727} C_VEL
LIN {X 0,Y 759.902,Z 781.063,A -85,B 0,C 180,E1 422.198,E2 422.198} C_VEL
LIN {X 0,Y 759.905,Z 758.091,A -85,B 0,C 180,E1 421.701,E2 421.701} C_VEL
LIN {X 0,Y 759.918,Z 735.874,A -85,B 0,C 180,E1 421.358,E2 421.358} C_VEL
LIN {X 0,Y 759.918,Z 462.428,A -85,B 0,C 180,E1 418.412,E2 418.412} C_VEL
LIN {X 0,Y 759.884,Z 347.462,A -85,B 0,C 180,E1 417.15,E2 417.15} C_VEL
LIN {X 0,Y 759.841,Z 326.577,A -85,B 0,C 180,E1 415.63,E2 415.63} C_VEL
LIN {X 0,Y 759.865,Z 326.576,A -85,B 0,C 180,E1 413.127,E2 413.127} C_VEL
LIN {X 0,Y 759.88,Z 326.57,A -85,B 0,C 180,E1 410.098,E2 410.098} C_VEL
LIN {X 0,Y 759.841,Z 326.573,A -85,B 0,C 180,E1 407.541,E2 407.541} C_VEL
LIN {X 0,Y 759.86,Z 326.574,A -85,B 0,C 180,E1 405.038,E2 405.038} C_VEL
LIN {X 0,Y 759.899,Z 326.568,A -85,B 0,C 180,E1 402.087,E2 402.087} C_VEL
LIN {X 0,Y 759.842,Z 326.572,A -85,B 0,C 180,E1 399.464,E2 399.464} C_VEL
LIN {X 0,Y 759.854,Z 326.575,A -85,B 0,C 180,E1 396.968,E2 396.968} C_VEL
LIN {X 0,Y 759.915,Z 326.569,A -85,B 0,C 180,E1 394.093,E2 394.093} C_VEL
LIN {X 0,Y 759.845,Z 326.572,A -85,B 0,C 180,E1 391.406,E2 391.406} C_VEL
LIN {X 0,Y 759.846,Z 326.574,A -85,B 0,C 180,E1 388.945,E2 388.945} C_VEL
LIN {X 0,Y 759.916,Z 326.574,A -85,B 0,C 180,E1 386.186,E2 386.186} C_VEL
LIN {X 0,Y 759.854,Z 326.571,A -85,B 0,C 180,E1 383.416,E2 383.416} C_VEL
LIN {X 0,Y 759.84,Z 326.573,A -85,B 0,C 180,E1 380.973,E2 380.973} C_VEL
LIN {X 0,Y 759.881,Z 326.576,A -85,B 0,C 180,E1 378.409,E2 378.409} C_VEL
LIN {X 0,Y 759.867,Z 326.57,A -85,B 0,C 180,E1 375.415,E2 375.415} C_VEL
LIN {X 0,Y 759.84,Z 326.573,A -85,B 0,C 180,E1 372.927,E2 372.927} C_VEL
LIN {X 0,Y 759.866,Z 326.575,A -85,B 0,C 180,E1 370.386,E2 370.386} C_VEL
LIN {X 0,Y 759.873,Z 326.57,A -85,B 0,C 180,E1 367.333,E2 367.333} C_VEL
LIN {X 0,Y 759.84,Z 326.573,A -85,B 0,C 180,E1 364.831,E2 364.831} C_VEL
LIN {X 0,Y 759.857,Z 326.575,A -85,B 0,C 180,E1 362.338,E2 362.338} C_VEL
LIN {X 0,Y 759.901,Z 326.569,A -85,B 0,C 180,E1 359.397,E2 359.397} C_VEL
LIN {X 0,Y 759.842,Z 326.572,A -85,B 0,C 180,E1 356.756,E2 356.756} C_VEL
LIN {X 0,Y 759.852,Z 326.575,A -85,B 0,C 180,E1 354.26,E2 354.26} C_VEL
LIN {X 0,Y 759.915,Z 326.569,A -85,B 0,C 180,E1 351.373,E2 351.373} C_VEL
LIN {X 0,Y 759.844,Z 326.572,A -85,B 0,C 180,E1 348.693,E2 348.693} C_VEL
LIN {X 0,Y 759.846,Z 326.574,A -85,B 0,C 180,E1 346.221,E2 346.221} C_VEL
LIN {X 0,Y 759.915,Z 326.575,A -85,B 0,C 180,E1 343.488,E2 343.488} C_VEL
LIN {X 0,Y 759.848,Z 326.572,A -85,B 0,C 180,E1 340.649,E2 340.649} C_VEL
LIN {X 0,Y 759.84,Z 326.573,A -85,B 0,C 180,E1 338.217,E2 338.217} C_VEL
LIN {X 0,Y 759.896,Z 326.577,A -85,B 0,C 180,E1 335.582,E2 335.582} C_VEL
LIN {X 0,Y 759.861,Z 326.571,A -85,B 0,C 180,E1 332.651,E2 332.651} C_VEL
LIN {X 0,Y 759.839,Z 326.573,A -85,B 0,C 180,E1 330.17,E2 330.17} C_VEL
LIN {X 0,Y 759.867,Z 326.576,A -85,B 0,C 180,E1 327.65,E2 327.65} C_VEL
LIN {X 0,Y 759.873,Z 326.57,A -85,B 0,C 180,E1 324.621,E2 324.621} C_VEL
LIN {X 0,Y 759.839,Z 326.573,A -85,B 0,C 180,E1 322.082,E2 322.082} C_VEL
LIN {X 0,Y 759.855,Z 326.575,A -85,B 0,C 180,E1 319.632,E2 319.632} C_VEL
LIN {X 0,Y 759.903,Z 326.569,A -85,B 0,C 180,E1 316.689,E2 316.689} C_VEL
LIN {X 0,Y 759.842,Z 326.572,A -85,B 0,C 180,E1 314.07,E2 314.07} C_VEL
LIN {X 0,Y 759.845,Z 326.575,A -85,B 0,C 180,E1 311.631,E2 311.631} C_VEL
LIN {X 0,Y 759.916,Z 326.573,A -85,B 0,C 180,E1 308.779,E2 308.779} C_VEL
LIN {X 0,Y 759.858,Z 326.711,A -85,B 0,C 180,E1 306.181,E2 306.181} C_VEL
LIN {X 0,Y 759.903,Z 363.722,A -85,B 0,C 180,E1 303.684,E2 303.684} C_VEL
LIN {X 0,Y 759.914,Z 377.341,A -85,B 0,C 180,E1 302.802,E2 302.802} C_VEL
LIN {X 0,Y 759.918,Z 632.42,A -85,B 0,C 180,E1 300.034,E2 300.034} C_VEL
LIN {X 0,Y 759.915,Z 765.99,A -85,B 0,C 180,E1 298.595,E2 298.595} C_VEL
LIN {X 0,Y 759.897,Z 790.298,A -85,B 0,C 180,E1 298.21,E2 298.21} C_VEL
LIN {X 0,Y 759.902,Z 811.681,A -85,B 0,C 180,E1 297.742,E2 297.742} C_VEL
LIN {X 0,Y 759.901,Z 831.085,A -85,B 0,C 180,E1 297.221,E2 297.221} C_VEL
LIN {X 0,Y 759.919,Z 853.737,A -85,B 0,C 180,E1 296.491,E2 296.491} C_VEL
LIN {X 0,Y 759.916,Z 875.25,A -85,B 0,C 180,E1 295.651,E2 295.651} C_VEL
LIN {X 0,Y 759.913,Z 894.66,A -85,B 0,C 180,E1 294.783,E2 294.783} C_VEL
LIN {X 0,Y 759.91,Z 917.06,A -85,B 0,C 180,E1 293.62,E2 293.62} C_VEL
LIN {X 0,Y 759.907,Z 935.705,A -85,B 0,C 180,E1 292.513,E2 292.513} C_VEL
LIN {X 0,Y 759.909,Z 955.523,A -85,B 0,C 180,E1 291.173,E2 291.173} C_VEL
LIN {X 0,Y 759.917,Z 972.885,A -85,B 0,C 180,E1 289.845,E2 289.845} C_VEL
LIN {X 0,Y 759.909,Z 989.39,A -85,B 0,C 180,E1 288.409,E2 288.409} C_VEL
LIN {X 0,Y 759.903,Z 1003.947,A -85,B 0,C 180,E1 286.984,E2 286.984} C_VEL
LIN {X 0,Y 759.915,Z 1018.836,A -85,B 0,C 180,E1 285.317,E2 285.317} C_VEL
LIN {X 0,Y 759.897,Z 1030.589,A -85,B 0,C 180,E1 283.812,E2 283.812} C_VEL
LIN {X 0,Y 759.901,Z 1042.785,A -85,B 0,C 180,E1 281.999,E2 281.999} C_VEL
LIN {X 0,Y 759.91,Z 1051.555,A -85,B 0,C 180,E1 280.462,E2 280.462} C_VEL
LIN {X 0,Y 759.89,Z 1060.073,A -85,B 0,C 180,E1 278.704,E2 278.704} C_VEL
LIN {X 0,Y 759.919,Z 1066.725,A -85,B 0,C 180,E1 276.953,E2 276.953} C_VEL
LIN {X 0,Y 759.906,Z 1071.51,A -85,B 0,C 180,E1 275.361,E2 275.361} C_VEL
LIN {X 0,Y 759.917,Z 1075.671,A -85,B 0,C 180,E1 273.395,E2 273.395} C_VEL
LIN {X 0,Y 759.899,Z 1077.63,A -85,B 0,C 180,E1 271.81,E2 271.81} C_VEL
LIN {X 0,Y 759.92,Z 1078.5,A -85,B 0,C 180,E1 270,E2 270} C_VEL
LIN {X 0,Y 759.899,Z 1077.63,A -85,B 0,C 180,E1 268.19,E2 268.19} C_VEL
LIN {X 0,Y 759.919,Z 1075.559,A -85,B 0,C 180,E1 266.53,E2 266.53} C_VEL
LIN {X 0,Y 759.906,Z 1071.51,A -85,B 0,C 180,E1 264.64,E2 264.64} C_VEL
LIN {X 0,Y 759.919,Z 1066.726,A -85,B 0,C 180,E1 263.047,E2 263.047} C_VEL
LIN {X 0,Y 759.892,Z 1059.73,A -85,B 0,C 180,E1 261.22,E2 261.22} C_VEL
LIN {X 0,Y 759.91,Z 1051.555,A -85,B 0,C 180,E1 259.538,E2 259.538} C_VEL
LIN {X 0,Y 759.901,Z 1042.786,A -85,B 0,C 180,E1 258.001,E2 258.001} C_VEL
LIN {X 0,Y 759.897,Z 1030.589,A -85,B 0,C 180,E1 256.188,E2 256.188} C_VEL
LIN {X 0,Y 759.917,Z 1018.833,A -85,B 0,C 180,E1 254.683,E2 254.683} C_VEL
LIN {X 0,Y 759.903,Z 1003.948,A -85,B 0,C 180,E1 253.016,E2 253.016} C_VEL
LIN {X 0,Y 759.909,Z 989.392,A -85,B 0,C 180,E1 251.591,E2 251.591} C_VEL
LIN {X 0,Y 759.911,Z 971.367,A -85,B 0,C 180,E1 250.035,E2 250.035} C_VEL
LIN {X 0,Y 759.913,Z 954.42,A -85,B 0,C 180,E1 248.746,E2 248.746} C_VEL
LIN {X 0,Y 759.909,Z 934.384,A -85,B 0,C 180,E1 247.405,E2 247.405} C_VEL
LIN {X 0,Y 759.91,Z 915.991,A -85,B 0,C 180,E1 246.32,E2 246.32} C_VEL
LIN {X 0,Y 759.912,Z 893.901,A -85,B 0,C 180,E1 245.182,E2 245.182} C_VEL
LIN {X 0,Y 759.916,Z 874.865,A -85,B 0,C 180,E1 244.332,E2 244.332} C_VEL
LIN {X 0,Y 759.916,Z 852.82,A -85,B 0,C 180,E1 243.475,E2 243.475} C_VEL
LIN {X 0,Y 759.901,Z 831.088,A -85,B 0,C 180,E1 242.779,E2 242.779} C_VEL
LIN {X 0,Y 759.902,Z 811.687,A -85,B 0,C 180,E1 242.258,E2 242.258} C_VEL
LIN {X 0,Y 759.899,Z 789.263,A -85,B 0,C 180,E1 241.768,E2 241.768} C_VEL
LIN {X 0,Y 759.917,Z 766.002,A -85,B 0,C 180,E1 241.405,E2 241.405} C_VEL
LIN {X 0,Y 759.899,Z 499.223,A -85,B 0,C 180,E1 238.53,E2 238.53} C_VEL
LIN {X 0,Y 759.911,Z 376.686,A -85,B 0,C 180,E1 237.173,E2 237.173} C_VEL
LIN {X 0,Y 759.853,Z 337.913,A -85,B 0,C 180,E1 234.582,E2 234.582} C_VEL
LIN {X 0,Y 759.861,Z 326.575,A -85,B 0,C 180,E1 233.784,E2 233.784} C_VEL
LIN {X 0,Y 759.888,Z 326.577,A -85,B 0,C 180,E1 230.808,E2 230.808} C_VEL
LIN {X 0,Y 759.841,Z 326.574,A -85,B 0,C 180,E1 228.252,E2 228.252} C_VEL
LIN {X 0,Y 759.85,Z 326.572,A -85,B 0,C 180,E1 225.779,E2 225.779} C_VEL
LIN {X 0,Y 759.913,Z 326.575,A -85,B 0,C 180,E1 222.968,E2 222.968} C_VEL
LIN {X 0,Y 759.848,Z 326.574,A -85,B 0,C 180,E1 220.249,E2 220.249} C_VEL
LIN {X 0,Y 759.842,Z 326.572,A -85,B 0,C 180,E1 217.823,E2 217.823} C_VEL
LIN {X 0,Y 759.9,Z 326.568,A -85,B 0,C 180,E1 215.193,E2 215.193} C_VEL
LIN {X 0,Y 759.864,Z 326.575,A -85,B 0,C 180,E1 212.293,E2 212.293} C_VEL
LIN {X 0,Y 759.841,Z 326.573,A -85,B 0,C 180,E1 209.83,E2 209.83} C_VEL
LIN {X 0,Y 759.863,Z 326.57,A -85,B 0,C 180,E1 207.338,E2 207.338} C_VEL
LIN {X 0,Y 759.898,Z 326.577,A -85,B 0,C 180,E1 204.404,E2 204.404} C_VEL
LIN {X 0,Y 759.843,Z 326.573,A -85,B 0,C 180,E1 201.783,E2 201.783} C_VEL
LIN {X 0,Y 759.854,Z 326.571,A -85,B 0,C 180,E1 199.287,E2 199.287} C_VEL
LIN {X 0,Y 759.914,Z 326.577,A -85,B 0,C 180,E1 196.355,E2 196.355} C_VEL
LIN {X 0,Y 759.846,Z 326.574,A -85,B 0,C 180,E1 193.702,E2 193.702} C_VEL
LIN {X 0,Y 759.851,Z 326.571,A -85,B 0,C 180,E1 191.23,E2 191.23} C_VEL
LIN {X 0,Y 759.915,Z 326.572,A -85,B 0,C 180,E1 188.475,E2 188.475} C_VEL
LIN {X 0,Y 759.852,Z 326.574,A -85,B 0,C 180,E1 185.664,E2 185.664} C_VEL
LIN {X 0,Y 759.848,Z 326.571,A -85,B 0,C 180,E1 183.168,E2 183.168} C_VEL
LIN {X 0,Y 759.918,Z 326.569,A -85,B 0,C 180,E1 180.452,E2 180.452} C_VEL
LIN {X 0,Y 759.857,Z 326.574,A -85,B 0,C 180,E1 177.587,E2 177.587} C_VEL
LIN {X 0,Y 759.845,Z 326.572,A -85,B 0,C 180,E1 177.165,E2 177.165} C_VEL
LIN {X 0,Y 758.857,Z 326.699,A -85,B 0,C 180,E1 176.584,E2 176.584} C_VEL
LIN {X 0,Y 752.445,Z 327.496,A -85,B 0,C 180,E1 174.958,E2 174.958} C_VEL
LIN {X 0,Y 751.958,Z 327.558,A -85,B 0,C 180,E1 174.535,E2 174.535} C_VEL
LIN {X 0,Y 751.929,Z 327.564,A -85,B 0,C 180,E1 171.589,E2 171.589} C_VEL
LIN {X 0,Y 751.907,Z 327.56,A -85,B 0,C 180,E1 169.038,E2 169.038} C_VEL
LIN {X 0,Y 751.961,Z 327.557,A -85,B 0,C 180,E1 166.387,E2 166.387} C_VEL
LIN {X 0,Y 751.932,Z 327.564,A -85,B 0,C 180,E1 163.467,E2 163.467} C_VEL
LIN {X 0,Y 751.908,Z 327.561,A -85,B 0,C 180,E1 160.905,E2 160.905} C_VEL
LIN {X 0,Y 751.965,Z 327.557,A -85,B 0,C 180,E1 158.223,E2 158.223} C_VEL
LIN {X 0,Y 751.923,Z 327.564,A -85,B 0,C 180,E1 155.236,E2 155.236} C_VEL
LIN {X 0,Y 751.91,Z 327.56,A -85,B 0,C 180,E1 152.691,E2 152.691} C_VEL
LIN {X 0,Y 751.978,Z 327.558,A -85,B 0,C 180,E1 149.914,E2 149.914} C_VEL
LIN {X 0,Y 751.92,Z 327.563,A -85,B 0,C 180,E1 147.044,E2 147.044} C_VEL
LIN {X 0,Y 751.915,Z 327.56,A -85,B 0,C 180,E1 144.47,E2 144.47} C_VEL
LIN {X 0,Y 751.976,Z 327.56,A -85,B 0,C 180,E1 141.676,E2 141.676} C_VEL
LIN {X 0,Y 751.924,Z 327.564,A -85,B 0,C 180,E1 138.935,E2 138.935} C_VEL
LIN {X 0,Y 751.914,Z 327.56,A -85,B 0,C 180,E1 136.357,E2 136.357} C_VEL
LIN {X 0,Y 751.978,Z 327.558,A -85,B 0,C 180,E1 133.638,E2 133.638} C_VEL
LIN {X 0,Y 751.922,Z 327.564,A -85,B 0,C 180,E1 130.762,E2 130.762} C_VEL
LIN {X 0,Y 751.916,Z 327.561,A -85,B 0,C 180,E1 128.195,E2 128.195} C_VEL
LIN {X 0,Y 751.975,Z 327.563,A -85,B 0,C 180,E1 125.403,E2 125.403} C_VEL
LIN {X 0,Y 751.937,Z 327.711,A -85,B 0,C 180,E1 124.585,E2 124.585} C_VEL
LIN {X 0,Y 752.678,Z 331.354,A -85,B 0,C 180,E1 124.28,E2 124.28} C_VEL
LIN {X 0,Y 752.762,Z 347.924,A -85,B 0,C 180,E1 123.102,E2 123.102} C_VEL
LIN {X 0,Y 753.146,Z 351.304,A -85,B 0,C 180,E1 123.045,E2 123.045} C_VEL
LIN {X 0,Y 752.992,Z 589.894,A -85,B 0,C 180,E1 120.43,E2 120.43} C_VEL
LIN {X 0,Y 752.882,Z 736.414,A -85,B 0,C 180,E1 118.837,E2 118.837} C_VEL
LIN {X 0,Y 752.8,Z 761.261,A -85,B 0,C 180,E1 118.435,E2 118.435} C_VEL
LIN {X 0,Y 752.755,Z 782.634,A -85,B 0,C 180,E1 117.96,E2 117.96} C_VEL
LIN {X 0,Y 752.691,Z 803.612,A -85,B 0,C 180,E1 117.385,E2 117.385} C_VEL
LIN {X 0,Y 752.616,Z 827.048,A -85,B 0,C 180,E1 116.598,E2 116.598} C_VEL
LIN {X 0,Y 752.546,Z 846.189,A -85,B 0,C 180,E1 115.836,E2 115.836} C_VEL
LIN {X 0,Y 752.459,Z 868.241,A -85,B 0,C 180,E1 114.829,E2 114.829} C_VEL
LIN {X 0,Y 752.364,Z 888.459,A -85,B 0,C 180,E1 113.746,E2 113.746} C_VEL
LIN {X 0,Y 752.299,Z 907.633,A -85,B 0,C 180,E1 112.589,E2 112.589} C_VEL
LIN {X 0,Y 752.202,Z 926.581,A -85,B 0,C 180,E1 111.278,E2 111.278} C_VEL
LIN {X 0,Y 752.145,Z 944.844,A -85,B 0,C 180,E1 109.855,E2 109.855} C_VEL
LIN {X 0,Y 752.086,Z 961.468,A -85,B 0,C 180,E1 108.366,E2 108.366} C_VEL
LIN {X 0,Y 752.015,Z 977.276,A -85,B 0,C 180,E1 106.77,E2 106.77} C_VEL
LIN {X 0,Y 751.992,Z 990.242,A -85,B 0,C 180,E1 105.264,E2 105.264} C_VEL
LIN {X 0,Y 751.969,Z 1003.01,A -85,B 0,C 180,E1 103.587,E2 103.587} C_VEL
LIN {X 0,Y 751.932,Z 1013.908,A -85,B 0,C 180,E1 101.895,E2 101.895} C_VEL
LIN {X 0,Y 751.933,Z 1022.543,A -85,B 0,C 180,E1 100.342,E2 100.342} C_VEL
LIN {X 0,Y 751.904,Z 1031.42,A -85,B 0,C 180,E1 98.411,E2 98.411} C_VEL
LIN {X 0,Y 751.914,Z 1037.34,A -85,B 0,C 180,E1 96.797,E2 96.797} C_VEL
LIN {X 0,Y 751.907,Z 1042.607,A -85,B 0,C 180,E1 94.959,E2 94.959} C_VEL
LIN {X 0,Y 751.91,Z 1046.055,A -85,B 0,C 180,E1 93.125,E2 93.125} C_VEL
LIN {X 0,Y 751.896,Z 1047.926,A -85,B 0,C 180,E1 91.448,E2 91.448} C_VEL
LIN {X 0,Y 751.89,Z 1048.386,A -85,B 0,C 180,E1 89.543,E2 89.543} C_VEL
LIN {X 0,Y 751.915,Z 1047.469,A -85,B 0,C 180,E1 87.942,E2 87.942} C_VEL
LIN {X 0,Y 751.914,Z 1044.857,A -85,B 0,C 180,E1 86.035,E2 86.035} C_VEL
LIN {X 0,Y 751.9,Z 1041.014,A -85,B 0,C 180,E1 84.353,E2 84.353} C_VEL
LIN {X 0,Y 751.908,Z 1036.112,A -85,B 0,C 180,E1 82.742,E2 82.742} C_VEL
LIN {X 0,Y 751.928,Z 1028.516,A -85,B 0,C 180,E1 80.818,E2 80.818} C_VEL
LIN {X 0,Y 751.913,Z 1020.976,A -85,B 0,C 180,E1 79.271,E2 79.271} C_VEL
LIN {X 0,Y 751.952,Z 1011.202,A -85,B 0,C 180,E1 77.56,E2 77.56} C_VEL
LIN {X 0,Y 751.973,Z 999.44,A -85,B 0,C 180,E1 75.838,E2 75.838} C_VEL
LIN {X 0,Y 751.998,Z 987.121,A -85,B 0,C 180,E1 74.261,E2 74.261} C_VEL
LIN {X 0,Y 752.05,Z 972.056,A -85,B 0,C 180,E1 72.593,E2 72.593} C_VEL
LIN {X 0,Y 752.075,Z 957.315,A -85,B 0,C 180,E1 71.151,E2 71.151} C_VEL
LIN {X 0,Y 752.161,Z 939.9,A -85,B 0,C 180,E1 69.658,E2 69.658} C_VEL
LIN {X 0,Y 752.225,Z 922.108,A -85,B 0,C 180,E1 68.302,E2 68.302} C_VEL
LIN {X 0,Y 752.312,Z 902.459,A -85,B 0,C 180,E1 66.999,E2 66.999} C_VEL
LIN {X 0,Y 752.408,Z 882.005,A -85,B 0,C 180,E1 65.797,E2 65.797} C_VEL
LIN {X 0,Y 752.486,Z 861.294,A -85,B 0,C 180,E1 64.752,E2 64.752} C_VEL
LIN {X 0,Y 752.557,Z 841.34,A -85,B 0,C 180,E1 63.867,E2 63.867} C_VEL
LIN {X 0,Y 752.643,Z 817.573,A -85,B 0,C 180,E1 62.977,E2 62.977} C_VEL
LIN {X 0,Y 752.713,Z 798.586,A -85,B 0,C 180,E1 62.379,E2 62.379} C_VEL
LIN {X 0,Y 752.771,Z 775.304,A -85,B 0,C 180,E1 61.768,E2 61.768} C_VEL
LIN {X 0,Y 752.843,Z 751.788,A -85,B 0,C 180,E1 61.306,E2 61.306} C_VEL
LIN {X 0,Y 752.884,Z 731.613,A -85,B 0,C 180,E1 61.012,E2 61.012} C_VEL
LIN {X 0,Y 753.092,Z 462.993,A -85,B 0,C 180,E1 58.099,E2 58.099} C_VEL
LIN {X 0,Y 752.944,Z 348.676,A -85,B 0,C 180,E1 56.826,E2 56.826} C_VEL
LIN {X 0,Y 752.673,Z 347.114,A -85,B 0,C 180,E1 56.771,E2 56.771} C_VEL
LIN {X 0,Y 752.628,Z 330.035,A -85,B 0,C 180,E1 55.531,E2 55.531} C_VEL
LIN {X 0,Y 751.914,Z 327.57,A -85,B 0,C 180,E1 55.309,E2 55.309} C_VEL
LIN {X 0,Y 751.978,Z 327.559,A -85,B 0,C 180,E1 52.387,E2 52.387} C_VEL
LIN {X 0,Y 751.908,Z 327.562,A -85,B 0,C 180,E1 49.738,E2 49.738} C_VEL
LIN {X 0,Y 751.91,Z 327.564,A -85,B 0,C 180,E1 47.227,E2 47.227} C_VEL
LIN {X 0,Y 751.976,Z 327.563,A -85,B 0,C 180,E1 44.435,E2 44.435} C_VEL
LIN {X 0,Y 751.91,Z 327.558,A -85,B 0,C 180,E1 41.639,E2 41.639} C_VEL
LIN {X 0,Y 751.906,Z 327.563,A -85,B 0,C 180,E1 39.17,E2 39.17} C_VEL
LIN {X 0,Y 751.977,Z 327.564,A -85,B 0,C 180,E1 36.373,E2 36.373} C_VEL
LIN {X 0,Y 751.909,Z 327.561,A -85,B 0,C 180,E1 33.495,E2 33.495} C_VEL
LIN {X 0,Y 751.904,Z 327.562,A -85,B 0,C 180,E1 31.062,E2 31.062} C_VEL
LIN {X 0,Y 751.979,Z 327.565,A -85,B 0,C 180,E1 28.328,E2 28.328} C_VEL
LIN {X 0,Y 751.913,Z 327.56,A -85,B 0,C 180,E1 25.437,E2 25.437} C_VEL
LIN {X 0,Y 751.904,Z 327.562,A -85,B 0,C 180,E1 22.932,E2 22.932} C_VEL
LIN {X 0,Y 751.979,Z 327.564,A -85,B 0,C 180,E1 20.144,E2 20.144} C_VEL
LIN {X 0,Y 751.911,Z 327.561,A -85,B 0,C 180,E1 17.25,E2 17.25} C_VEL
LIN {X 0,Y 751.903,Z 327.562,A -85,B 0,C 180,E1 14.793,E2 14.793} C_VEL
LIN {X 0,Y 751.973,Z 327.566,A -85,B 0,C 180,E1 12.05,E2 12.05} C_VEL
LIN {X 0,Y 751.915,Z 327.56,A -85,B 0,C 180,E1 9.182,E2 9.182} C_VEL
LIN {X 0,Y 751.903,Z 327.562,A -85,B 0,C 180,E1 6.72,E2 6.72} C_VEL
LIN {X 0,Y 751.961,Z 327.566,A -85,B 0,C 180,E1 4.041,E2 4.041} C_VEL
LIN {X 0,Y 751.917,Z 327.559,A -85,B 0,C 180,E1 1.067,E2 1.067} C_VEL
LIN {X 0,Y 751.901,Z 327.562,A -85,B 0,C 180,E1 -1.372,E2 -1.372} C_VEL
LIN {X 0,Y 751.941,Z 327.564,A -85,B 0,C 180,E1 -3.965,E2 -3.965} C_VEL
LIN {X 0,Y 751.929,Z 327.559,A -85,B 0,C 180,E1 -6.95,E2 -6.95} C_VEL
LIN {X 0,Y 751.901,Z 327.562,A -85,B 0,C 180,E1 -9.491,E2 -9.491} C_VEL
LIN {X 0,Y 751.934,Z 327.565,A -85,B 0,C 180,E1 -12.05,E2 -12.05} C_VEL
LIN {X 0,Y 751.926,Z 327.559,A -85,B 0,C 180,E1 -15.113,E2 -15.113} C_VEL
LIN {X 0,Y 751.9,Z 327.562,A -85,B 0,C 180,E1 -17.65,E2 -17.65} C_VEL
LIN {X 0,Y 751.929,Z 327.565,A -85,B 0,C 180,E1 -20.146,E2 -20.146} C_VEL
LIN {X 0,Y 751.927,Z 327.559,A -85,B 0,C 180,E1 -23.238,E2 -23.238} C_VEL
LIN {X 0,Y 751.901,Z 327.562,A -85,B 0,C 180,E1 -25.691,E2 -25.691} C_VEL
LIN {X 0,Y 751.916,Z 327.564,A -85,B 0,C 180,E1 -28.169,E2 -28.169} C_VEL
LIN {X 0,Y 751.964,Z 327.558,A -85,B 0,C 180,E1 -31.093,E2 -31.093} C_VEL
LIN {X 0,Y 751.902,Z 327.562,A -85,B 0,C 180,E1 -33.785,E2 -33.785} C_VEL
LIN {X 0,Y 751.917,Z 327.564,A -85,B 0,C 180,E1 -36.307,E2 -36.307} C_VEL
LIN {X 0,Y 751.96,Z 327.558,A -85,B 0,C 180,E1 -39.268,E2 -39.268} C_VEL
LIN {X 0,Y 751.902,Z 327.561,A -85,B 0,C 180,E1 -41.88,E2 -41.88} C_VEL
LIN {X 0,Y 751.908,Z 327.564,A -85,B 0,C 180,E1 -44.321,E2 -44.321} C_VEL
LIN {X 0,Y 751.978,Z 327.563,A -85,B 0,C 180,E1 -47.11,E2 -47.11} C_VEL
LIN {X 0,Y 751.91,Z 327.562,A -85,B 0,C 180,E1 -49.875,E2 -49.875} C_VEL
LIN {X 0,Y 751.901,Z 327.565,A -85,B 0,C 180,E1 -52.302,E2 -52.302} C_VEL
LIN {X 0,Y 751.991,Z 327.722,A -85,B 0,C 180,E1 -53.449,E2 -53.449} C_VEL
LIN {X 0,Y 752.812,Z 331.087,A -85,B 0,C 180,E1 -53.729,E2 -53.729} C_VEL
LIN {X 0,Y 752.744,Z 367.133,A -85,B 0,C 180,E1 -56.181,E2 -56.181} C_VEL
LIN {X 0,Y 752.801,Z 377.401,A -85,B 0,C 180,E1 -56.849,E2 -56.849} C_VEL
LIN {X 0,Y 753.183,Z 380.844,A -85,B 0,C 180,E1 -56.907,E2 -56.907} C_VEL
LIN {X 0,Y 752.979,Z 638.156,A -85,B 0,C 180,E1 -59.722,E2 -59.722} C_VEL
LIN {X 0,Y 752.879,Z 766.525,A -85,B 0,C 180,E1 -61.119,E2 -61.119} C_VEL
LIN {X 0,Y 752.8,Z 791.573,A -85,B 0,C 180,E1 -61.526,E2 -61.526} C_VEL
LIN {X 0,Y 752.755,Z 812.706,A -85,B 0,C 180,E1 -61.997,E2 -61.997} C_VEL
LIN {X 0,Y 752.694,Z 833.68,A -85,B 0,C 180,E1 -62.572,E2 -62.572} C_VEL
LIN {X 0,Y 752.614,Z 857.108,A -85,B 0,C 180,E1 -63.36,E2 -63.36} C_VEL
LIN {X 0,Y 752.545,Z 876.247,A -85,B 0,C 180,E1 -64.121,E2 -64.121} C_VEL
LIN {X 0,Y 752.469,Z 897.461,A -85,B 0,C 180,E1 -65.087,E2 -65.087} C_VEL
LIN {X 0,Y 752.363,Z 918.517,A -85,B 0,C 180,E1 -66.212,E2 -66.212} C_VEL
LIN {X 0,Y 752.292,Z 938.353,A -85,B 0,C 180,E1 -67.411,E2 -67.411} C_VEL
LIN {X 0,Y 752.2,Z 957.679,A -85,B 0,C 180,E1 -68.759,E2 -68.759} C_VEL
LIN {X 0,Y 752.131,Z 975.815,A -85,B 0,C 180,E1 -70.184,E2 -70.184} C_VEL
LIN {X 0,Y 752.084,Z 991.943,A -85,B 0,C 180,E1 -71.634,E2 -71.634} C_VEL
LIN {X 0,Y 752.018,Z 1007.675,A -85,B 0,C 180,E1 -73.23,E2 -73.23} C_VEL
LIN {X 0,Y 751.997,Z 1020.606,A -85,B 0,C 180,E1 -74.736,E2 -74.736} C_VEL
LIN {X 0,Y 751.967,Z 1033.325,A -85,B 0,C 180,E1 -76.413,E2 -76.413} C_VEL
LIN {X 0,Y 751.924,Z 1044.174,A -85,B 0,C 180,E1 -78.105,E2 -78.105} C_VEL
LIN {X 0,Y 751.931,Z 1052.779,A -85,B 0,C 180,E1 -79.658,E2 -79.658} C_VEL
LIN {X 0,Y 751.904,Z 1061.597,A -85,B 0,C 180,E1 -81.589,E2 -81.589} C_VEL
LIN {X 0,Y 751.906,Z 1067.488,A -85,B 0,C 180,E1 -83.203,E2 -83.203} C_VEL
LIN {X 0,Y 751.916,Z 1072.701,A -85,B 0,C 180,E1 -85.041,E2 -85.041} C_VEL
LIN {X 0,Y 751.916,Z 1076.121,A -85,B 0,C 180,E1 -86.875,E2 -86.875} C_VEL
LIN {X 0,Y 751.903,Z 1078.099,A -85,B 0,C 180,E1 -88.705,E2 -88.705} C_VEL
LIN {X 0,Y 751.891,Z 1078.351,A -85,B 0,C 180,E1 -90.533,E2 -90.533} C_VEL
LIN {X 0,Y 751.913,Z 1077.296,A -85,B 0,C 180,E1 -92.21,E2 -92.21} C_VEL
LIN {X 0,Y 751.91,Z 1074.343,A -85,B 0,C 180,E1 -94.168,E2 -94.168} C_VEL
LIN {X 0,Y 751.916,Z 1070.687,A -85,B 0,C 180,E1 -95.724,E2 -95.724} C_VEL
LIN {X 0,Y 751.897,Z 1064.936,A -85,B 0,C 180,E1 -97.565,E2 -97.565} C_VEL
LIN {X 0,Y 751.919,Z 1057.524,A -85,B 0,C 180,E1 -99.353,E2 -99.353} C_VEL
LIN {X 0,Y 751.924,Z 1049.517,A -85,B 0,C 180,E1 -100.962,E2 -100.962} C_VEL
LIN {X 0,Y 751.948,Z 1038.35,A -85,B 0,C 180,E1 -102.83,E2 -102.83} C_VEL
LIN {X 0,Y 751.97,Z 1027.951,A -85,B 0,C 180,E1 -104.319,E2 -104.319} C_VEL
LIN {X 0,Y 751.999,Z 1014.677,A -85,B 0,C 180,E1 -105.984,E2 -105.984} C_VEL
LIN {X 0,Y 752.053,Z 1000.842,A -85,B 0,C 180,E1 -107.486,E2 -107.486} C_VEL
LIN {X 0,Y 752.108,Z 984.651,A -85,B 0,C 180,E1 -109.048,E2 -109.048} C_VEL
LIN {X 0,Y 752.164,Z 967.821,A -85,B 0,C 180,E1 -110.464,E2 -110.464} C_VEL
LIN {X 0,Y 752.242,Z 948.444,A -85,B 0,C 180,E1 -111.906,E2 -111.906} C_VEL
LIN {X 0,Y 752.311,Z 930.418,A -85,B 0,C 180,E1 -113.084,E2 -113.084} C_VEL
LIN {X 0,Y 752.415,Z 908.749,A -85,B 0,C 180,E1 -114.328,E2 -114.328} C_VEL
LIN {X 0,Y 752.489,Z 889.455,A -85,B 0,C 180,E1 -115.29,E2 -115.29} C_VEL
LIN {X 0,Y 752.594,Z 867.168,A -85,B 0,C 180,E1 -116.259,E2 -116.259} C_VEL
LIN {X 0,Y 752.645,Z 846.237,A -85,B 0,C 180,E1 -117.023,E2 -117.023} C_VEL
LIN {X 0,Y 752.718,Z 827.021,A -85,B 0,C 180,E1 -117.621,E2 -117.621} C_VEL
LIN {X 0,Y 752.782,Z 802.765,A -85,B 0,C 180,E1 -118.242,E2 -118.242} C_VEL
LIN {X 0,Y 752.842,Z 781.052,A -85,B 0,C 180,E1 -118.661,E2 -118.661} C_VEL
LIN {X 0,Y 752.883,Z 760.649,A -85,B 0,C 180,E1 -118.955,E2 -118.955} C_VEL
LIN {X 0,Y 753.066,Z 501.64,A -85,B 0,C 180,E1 -121.762,E2 -121.762} C_VEL
LIN {X 0,Y 753.009,Z 378.268,A -85,B 0,C 180,E1 -123.131,E2 -123.131} C_VEL
LIN {X 0,Y 752.714,Z 376.594,A -85,B 0,C 180,E1 -123.187,E2 -123.187} C_VEL
LIN {X 0,Y 752.785,Z 339.846,A -85,B 0,C 180,E1 -125.669,E2 -125.669} C_VEL
LIN {X 0,Y 752.792,Z 330.295,A -85,B 0,C 180,E1 -126.327,E2 -126.327} C_VEL
LIN {X 0,Y 751.974,Z 327.564,A -85,B 0,C 180,E1 -126.569,E2 -126.569} C_VEL
LIN {X 0,Y 751.916,Z 327.566,A -85,B 0,C 180,E1 -129.467,E2 -129.467} C_VEL
LIN {X 0,Y 751.902,Z 327.562,A -85,B 0,C 180,E1 -131.982,E2 -131.982} C_VEL
LIN {X 0,Y 751.97,Z 327.559,A -85,B 0,C 180,E1 -134.701,E2 -134.701} C_VEL
LIN {X 0,Y 751.917,Z 327.564,A -85,B 0,C 180,E1 -137.607,E2 -137.607} C_VEL
LIN {X 0,Y 751.902,Z 327.561,A -85,B 0,C 180,E1 -140.112,E2 -140.112} C_VEL
LIN {X 0,Y 751.965,Z 327.558,A -85,B 0,C 180,E1 -142.796,E2 -142.796} C_VEL
LIN {X 0,Y 751.924,Z 327.564,A -85,B 0,C 180,E1 -145.679,E2 -145.679} C_VEL
LIN {X 0,Y 751.901,Z 327.561,A -85,B 0,C 180,E1 -148.223,E2 -148.223} C_VEL
LIN {X 0,Y 751.942,Z 327.559,A -85,B 0,C 180,E1 -150.79,E2 -150.79} C_VEL
LIN {X 0,Y 751.928,Z 327.564,A -85,B 0,C 180,E1 -153.801,E2 -153.801} C_VEL
LIN {X 0,Y 751.903,Z 327.561,A -85,B 0,C 180,E1 -156.321,E2 -156.321} C_VEL
LIN {X 0,Y 751.937,Z 327.559,A -85,B 0,C 180,E1 -158.877,E2 -158.877} C_VEL
LIN {X 0,Y 751.927,Z 327.564,A -85,B 0,C 180,E1 -161.949,E2 -161.949} C_VEL
LIN {X 0,Y 751.904,Z 327.561,A -85,B 0,C 180,E1 -164.497,E2 -164.497} C_VEL
LIN {X 0,Y 751.96,Z 327.558,A -85,B 0,C 180,E1 -167.17,E2 -167.17} C_VEL
LIN {X 0,Y 751.923,Z 327.564,A -85,B 0,C 180,E1 -170.123,E2 -170.123} C_VEL
LIN {X 0,Y 751.905,Z 327.56,A -85,B 0,C 180,E1 -172.665,E2 -172.665} C_VEL
LIN {X 0,Y 751.966,Z 327.558,A -85,B 0,C 180,E1 -175.348,E2 -175.348} C_VEL
LIN {X 0,Y 751.92,Z 327.564,A -85,B 0,C 180,E1 -178.324,E2 -178.324} C_VEL
LIN {X 0,Y 751.907,Z 327.561,A -85,B 0,C 180,E1 -180.838,E2 -180.838} C_VEL
LIN {X 0,Y 751.974,Z 327.557,A -85,B 0,C 180,E1 -183.583,E2 -183.583} C_VEL
LIN {X 0,Y 751.958,Z 327.558,A -85,B 0,C 180,E1 -185.465,E2 -185.465} C_VEL
LIN {X 0,Y 751.038,Z 327.682,A -85,B 0,C 180,E1 -186.051,E2 -186.051} C_VEL
LIN {X 0,Y 744.516,Z 328.502,A -85,B 0,C 180,E1 -187.736,E2 -187.736} C_VEL
LIN {X 0,Y 744.029,Z 328.555,A -85,B 0,C 180,E1 -188.121,E2 -188.121} C_VEL
LIN {X 0,Y 743.968,Z 328.549,A -85,B 0,C 180,E1 -190.845,E2 -190.845} C_VEL
LIN {X 0,Y 743.998,Z 328.547,A -85,B 0,C 180,E1 -193.444,E2 -193.444} C_VEL
LIN {X 0,Y 743.999,Z 328.554,A -85,B 0,C 180,E1 -196.474,E2 -196.474} C_VEL
LIN {X 0,Y 743.969,Z 328.55,A -85,B 0,C 180,E1 -199.062,E2 -199.062} C_VEL
LIN {X 0,Y 744.013,Z 328.546,A -85,B 0,C 180,E1 -201.69,E2 -201.69} C_VEL
LIN {X 0,Y 743.99,Z 328.553,A -85,B 0,C 180,E1 -204.707,E2 -204.707} C_VEL
LIN {X 0,Y 743.971,Z 328.549,A -85,B 0,C 180,E1 -207.278,E2 -207.278} C_VEL
LIN {X 0,Y 744.038,Z 328.546,A -85,B 0,C 180,E1 -209.995,E2 -209.995} C_VEL
LIN {X 0,Y 743.987,Z 328.553,A -85,B 0,C 180,E1 -212.886,E2 -212.886} C_VEL
LIN {X 0,Y 743.974,Z 328.549,A -85,B 0,C 180,E1 -215.493,E2 -215.493} C_VEL
LIN {X 0,Y 744.037,Z 328.548,A -85,B 0,C 180,E1 -218.296,E2 -218.296} C_VEL
LIN {X 0,Y 743.983,Z 328.553,A -85,B 0,C 180,E1 -221.087,E2 -221.087} C_VEL
LIN {X 0,Y 743.978,Z 328.549,A -85,B 0,C 180,E1 -223.692,E2 -223.692} C_VEL
LIN {X 0,Y 744.037,Z 328.551,A -85,B 0,C 180,E1 -226.527,E2 -226.527} C_VEL
LIN {X 0,Y 743.978,Z 328.553,A -85,B 0,C 180,E1 -229.32,E2 -229.32} C_VEL
LIN {X 0,Y 743.984,Z 328.55,A -85,B 0,C 180,E1 -231.911,E2 -231.911} C_VEL
LIN {X 0,Y 744.038,Z 328.555,A -85,B 0,C 180,E1 -234.794,E2 -234.794} C_VEL
LIN {X 0,Y 744.047,Z 328.815,A -85,B 0,C 180,E1 -235.077,E2 -235.077} C_VEL
LIN {X 0,Y 745.507,Z 333.868,A -85,B 0,C 180,E1 -235.529,E2 -235.529} C_VEL
LIN {X 0,Y 745.582,Z 347.978,A -85,B 0,C 180,E1 -236.538,E2 -236.538} C_VEL
LIN {X 0,Y 746.434,Z 352.26,A -85,B 0,C 180,E1 -236.629,E2 -236.629} C_VEL
LIN {X 0,Y 746.09,Z 590.709,A -85,B 0,C 180,E1 -239.267,E2 -239.267} C_VEL
LIN {X 0,Y 745.865,Z 736.458,A -85,B 0,C 180,E1 -240.866,E2 -240.866} C_VEL
LIN {X 0,Y 745.723,Z 761.385,A -85,B 0,C 180,E1 -241.272,E2 -241.272} C_VEL
LIN {X 0,Y 745.624,Z 782.894,A -85,B 0,C 180,E1 -241.755,E2 -241.755} C_VEL
LIN {X 0,Y 745.499,Z 805.102,A -85,B 0,C 180,E1 -242.372,E2 -242.372} C_VEL
LIN {X 0,Y 745.325,Z 828.073,A -85,B 0,C 180,E1 -243.16,E2 -243.16} C_VEL
LIN {X 0,Y 745.183,Z 848.193,A -85,B 0,C 180,E1 -243.975,E2 -243.975} C_VEL
LIN {X 0,Y 744.968,Z 871.482,A -85,B 0,C 180,E1 -245.074,E2 -245.074} C_VEL
LIN {X 0,Y 744.821,Z 890.578,A -85,B 0,C 180,E1 -246.12,E2 -246.12} C_VEL
LIN {X 0,Y 744.64,Z 911.374,A -85,B 0,C 180,E1 -247.416,E2 -247.416} C_VEL
LIN {X 0,Y 744.492,Z 929.344,A -85,B 0,C 180,E1 -248.697,E2 -248.697} C_VEL
LIN {X 0,Y 744.333,Z 948.093,A -85,B 0,C 180,E1 -250.213,E2 -250.213} C_VEL
LIN {X 0,Y 744.257,Z 963.175,A -85,B 0,C 180,E1 -251.596,E2 -251.596} C_VEL
LIN {X 0,Y 744.13,Z 979.404,A -85,B 0,C 180,E1 -253.289,E2 -253.289} C_VEL
LIN {X 0,Y 744.067,Z 992.172,A -85,B 0,C 180,E1 -254.809,E2 -254.809} C_VEL
LIN {X 0,Y 744.002,Z 1005.617,A -85,B 0,C 180,E1 -256.659,E2 -256.659} C_VEL
LIN {X 0,Y 743.961,Z 1015.3,A -85,B 0,C 180,E1 -258.212,E2 -258.212} C_VEL
LIN {X 0,Y 743.93,Z 1024.91,A -85,B 0,C 180,E1 -260.015,E2 -260.015} C_VEL
LIN {X 0,Y 743.921,Z 1032.334,A -85,B 0,C 180,E1 -261.731,E2 -261.731} C_VEL
LIN {X 0,Y 743.91,Z 1038.104,A -85,B 0,C 180,E1 -263.362,E2 -263.362} C_VEL
LIN {X 0,Y 743.907,Z 1043.244,A -85,B 0,C 180,E1 -265.297,E2 -265.297} C_VEL
LIN {X 0,Y 743.91,Z 1046.168,A -85,B 0,C 180,E1 -266.918,E2 -266.918} C_VEL
LIN {X 0,Y 743.908,Z 1048.125,A -85,B 0,C 180,E1 -268.768,E2 -268.768} C_VEL
LIN {X 0,Y 743.893,Z 1048.341,A -85,B 0,C 180,E1 -270.616,E2 -270.616} C_VEL
LIN {X 0,Y 743.916,Z 1047.269,A -85,B 0,C 180,E1 -272.311,E2 -272.311} C_VEL
LIN {X 0,Y 743.913,Z 1044.38,A -85,B 0,C 180,E1 -274.24,E2 -274.24} C_VEL
LIN {X 0,Y 743.918,Z 1040.601,A -85,B 0,C 180,E1 -275.863,E2 -275.863} C_VEL
LIN {X 0,Y 743.902,Z 1034.812,A -85,B 0,C 180,E1 -277.725,E2 -277.725} C_VEL
LIN {X 0,Y 743.926,Z 1027.45,A -85,B 0,C 180,E1 -279.516,E2 -279.516} C_VEL
LIN {X 0,Y 743.948,Z 1019.751,A -85,B 0,C 180,E1 -281.081,E2 -281.081} C_VEL
LIN {X 0,Y 743.984,Z 1008.47,A -85,B 0,C 180,E1 -282.997,E2 -282.997} C_VEL
LIN {X 0,Y 744.043,Z 997.7,A -85,B 0,C 180,E1 -284.555,E2 -284.555} C_VEL
LIN {X 0,Y 744.124,Z 983.733,A -85,B 0,C 180,E1 -286.31,E2 -286.31} C_VEL
LIN {X 0,Y 744.184,Z 969.721,A -85,B 0,C 180,E1 -287.839,E2 -287.839} C_VEL
LIN {X 0,Y 744.327,Z 952.83,A -85,B 0,C 180,E1 -289.46,E2 -289.46} C_VEL
LIN {X 0,Y 744.433,Z 936.346,A -85,B 0,C 180,E1 -290.851,E2 -290.851} C_VEL
LIN {X 0,Y 744.599,Z 916.868,A -85,B 0,C 180,E1 -292.296,E2 -292.296} C_VEL
LIN {X 0,Y 744.74,Z 898.357,A -85,B 0,C 180,E1 -293.508,E2 -293.508} C_VEL
LIN {X 0,Y 744.94,Z 877.402,A -85,B 0,C 180,E1 -294.704,E2 -294.704} C_VEL
LIN {X 0,Y 745.082,Z 857.725,A -85,B 0,C 180,E1 -295.687,E2 -295.687} C_VEL
LIN {X 0,Y 745.301,Z 833.875,A -85,B 0,C 180,E1 -296.707,E2 -296.707} C_VEL
LIN {X 0,Y 745.41,Z 813.741,A -85,B 0,C 180,E1 -297.437,E2 -297.437} C_VEL
LIN {X 0,Y 745.615,Z 790.309,A -85,B 0,C 180,E1 -298.148,E2 -298.148} C_VEL
LIN {X 0,Y 745.709,Z 767.509,A -85,B 0,C 180,E1 -298.69,E2 -298.69} C_VEL
LIN {X 0,Y 745.814,Z 746.983,A -85,B 0,C 180,E1 -299.071,E2 -299.071} C_VEL
LIN {X 0,Y 745.905,Z 716.267,A -85,B 0,C 180,E1 -299.463,E2 -299.463} C_VEL
LIN {X 0,Y 746.293,Z 460.943,A -85,B 0,C 180,E1 -302.249,E2 -302.249} C_VEL
LIN {X 0,Y 746.26,Z 350.489,A -85,B 0,C 180,E1 -303.489,E2 -303.489} C_VEL
LIN {X 0,Y 745.478,Z 347.264,A -85,B 0,C 180,E1 -303.581,E2 -303.581} C_VEL
LIN {X 0,Y 745.406,Z 333.171,A -85,B 0,C 180,E1 -304.618,E2 -304.618} C_VEL
LIN {X 0,Y 744.013,Z 328.557,A -85,B 0,C 180,E1 -305.043,E2 -305.043} C_VEL
LIN {X 0,Y 743.983,Z 328.551,A -85,B 0,C 180,E1 -308.041,E2 -308.041} C_VEL
LIN {X 0,Y 743.966,Z 328.553,A -85,B 0,C 180,E1 -310.592,E2 -310.592} C_VEL
LIN {X 0,Y 744.024,Z 328.554,A -85,B 0,C 180,E1 -313.266,E2 -313.266} C_VEL
LIN {X 0,Y 743.981,Z 328.55,A -85,B 0,C 180,E1 -316.199,E2 -316.199} C_VEL
LIN {X 0,Y 743.964,Z 328.548,A -85,B 0,C 180,E1 -318.707,E2 -318.707} C_VEL
LIN {X 0,Y 744.017,Z 328.554,A -85,B 0,C 180,E1 -321.335,E2 -321.335} C_VEL
LIN {X 0,Y 743.983,Z 328.549,A -85,B 0,C 180,E1 -324.318,E2 -324.318} C_VEL
LIN {X 0,Y 743.965,Z 328.551,A -85,B 0,C 180,E1 -326.858,E2 -326.858} C_VEL
LIN {X 0,Y 744.036,Z 328.554,A -85,B 0,C 180,E1 -329.629,E2 -329.629} C_VEL
LIN {X 0,Y 743.978,Z 328.548,A -85,B 0,C 180,E1 -332.502,E2 -332.502} C_VEL
LIN {X 0,Y 743.962,Z 328.552,A -85,B 0,C 180,E1 -334.953,E2 -334.953} C_VEL
LIN {X 0,Y 744.022,Z 328.554,A -85,B 0,C 180,E1 -337.646,E2 -337.646} C_VEL
LIN {X 0,Y 743.98,Z 328.548,A -85,B 0,C 180,E1 -340.612,E2 -340.612} C_VEL
LIN {X 0,Y 743.964,Z 328.552,A -85,B 0,C 180,E1 -343.124,E2 -343.124} C_VEL
LIN {X 0,Y 744.03,Z 328.554,A -85,B 0,C 180,E1 -345.842,E2 -345.842} C_VEL
LIN {X 0,Y 743.978,Z 328.547,A -85,B 0,C 180,E1 -348.762,E2 -348.762} C_VEL
LIN {X 0,Y 743.964,Z 328.552,A -85,B 0,C 180,E1 -351.265,E2 -351.265} C_VEL
LIN {X 0,Y 744.029,Z 328.554,A -85,B 0,C 180,E1 -353.983,E2 -353.983} C_VEL
LIN {X 0,Y 743.978,Z 328.549,A -85,B 0,C 180,E1 -356.918,E2 -356.918} C_VEL
LIN {X 0,Y 743.964,Z 328.55,A -85,B 0,C 180,E1 -359.384,E2 -359.384} C_VEL
LIN {X 0,Y 744.024,Z 328.555,A -85,B 0,C 180,E1 -362.079,E2 -362.079} C_VEL
LIN {X 0,Y 743.981,Z 328.549,A -85,B 0,C 180,E1 -365.012,E2 -365.012} C_VEL
LIN {X 0,Y 743.962,Z 328.55,A -85,B 0,C 180,E1 -367.491,E2 -367.491} C_VEL
LIN {X 0,Y 744.012,Z 328.554,A -85,B 0,C 180,E1 -370.14,E2 -370.14} C_VEL
LIN {X 0,Y 743.982,Z 328.548,A -85,B 0,C 180,E1 -373.128,E2 -373.128} C_VEL
LIN {X 0,Y 743.964,Z 328.551,A -85,B 0,C 180,E1 -375.673,E2 -375.673} C_VEL
LIN {X 0,Y 744.033,Z 328.555,A -85,B 0,C 180,E1 -378.418,E2 -378.418} C_VEL
LIN {X 0,Y 743.974,Z 328.549,A -85,B 0,C 180,E1 -381.36,E2 -381.36} C_VEL
LIN {X 0,Y 743.964,Z 328.552,A -85,B 0,C 180,E1 -383.863,E2 -383.863} C_VEL
LIN {X 0,Y 744.031,Z 328.556,A -85,B 0,C 180,E1 -386.584,E2 -386.584} C_VEL
LIN {X 0,Y 743.976,Z 328.55,A -85,B 0,C 180,E1 -389.466,E2 -389.466} C_VEL
LIN {X 0,Y 743.963,Z 328.551,A -85,B 0,C 180,E1 -391.974,E2 -391.974} C_VEL
LIN {X 0,Y 744.039,Z 328.554,A -85,B 0,C 180,E1 -394.736,E2 -394.736} C_VEL
LIN {X 0,Y 743.976,Z 328.55,A -85,B 0,C 180,E1 -397.602,E2 -397.602} C_VEL
LIN {X 0,Y 743.964,Z 328.551,A -85,B 0,C 180,E1 -400.116,E2 -400.116} C_VEL
LIN {X 0,Y 744.029,Z 328.556,A -85,B 0,C 180,E1 -402.844,E2 -402.844} C_VEL
LIN {X 0,Y 743.975,Z 328.55,A -85,B 0,C 180,E1 -405.754,E2 -405.754} C_VEL
LIN {X 0,Y 743.963,Z 328.553,A -85,B 0,C 180,E1 -408.239,E2 -408.239} C_VEL
LIN {X 0,Y 744.04,Z 328.555,A -85,B 0,C 180,E1 -411.029,E2 -411.029} C_VEL
LIN {X 0,Y 744.045,Z 328.587,A -85,B 0,C 180,E1 -413.056,E2 -413.056} C_VEL
LIN {X 0,Y 745.779,Z 334.386,A -85,B 0,C 180,E1 -413.563,E2 -413.563} C_VEL
LIN {X 0,Y 745.596,Z 369.861,A -85,B 0,C 180,E1 -415.998,E2 -415.998} C_VEL
LIN {X 0,Y 745.658,Z 377.521,A -85,B 0,C 180,E1 -416.492,E2 -416.492} C_VEL
LIN {X 0,Y 746.472,Z 381.891,A -85,B 0,C 180,E1 -416.582,E2 -416.582} C_VEL
LIN {X 0,Y 746.061,Z 639.683,A -85,B 0,C 180,E1 -419.428,E2 -419.428} C_VEL
LIN {X 0,Y 745.862,Z 766.633,A -85,B 0,C 180,E1 -420.823,E2 -420.823} C_VEL
LIN {X 0,Y 745.723,Z 791.759,A -85,B 0,C 180,E1 -421.235,E2 -421.235} C_VEL
LIN {X 0,Y 745.624,Z 813.032,A -85,B 0,C 180,E1 -421.713,E2 -421.713} C_VEL
LIN {X 0,Y 745.502,Z 835.078,A -85,B 0,C 180,E1 -422.326,E2 -422.326} C_VEL
LIN {X 0,Y 745.321,Z 858.807,A -85,B 0,C 180,E1 -423.143,E2 -423.143} C_VEL
LIN {X 0,Y 745.177,Z 879.234,A -85,B 0,C 180,E1 -423.974,E2 -423.974} C_VEL
LIN {X 0,Y 744.962,Z 902.332,A -85,B 0,C 180,E1 -425.074,E2 -425.074} C_VEL
LIN {X 0,Y 744.818,Z 921.355,A -85,B 0,C 180,E1 -426.12,E2 -426.12} C_VEL
LIN {X 0,Y 744.619,Z 943.231,A -85,B 0,C 180,E1 -427.499,E2 -427.499} C_VEL
LIN {X 0,Y 744.489,Z 960.817,A -85,B 0,C 180,E1 -428.762,E2 -428.762} C_VEL
LIN {X 0,Y 744.337,Z 978.602,A -85,B 0,C 180,E1 -430.213,E2 -430.213} C_VEL
LIN {X 0,Y 744.244,Z 994.495,A -85,B 0,C 180,E1 -431.677,E2 -431.677} C_VEL
LIN {X 0,Y 744.132,Z 1009.799,A -85,B 0,C 180,E1 -433.289,E2 -433.289} C_VEL
LIN {X 0,Y 744.067,Z 1023.175,A -85,B 0,C 180,E1 -434.888,E2 -434.888} C_VEL
LIN {X 0,Y 744.007,Z 1035.901,A -85,B 0,C 180,E1 -436.658,E2 -436.658} C_VEL
LIN {X 0,Y 743.953,Z 1045.563,A -85,B 0,C 180,E1 -438.212,E2 -438.212} C_VEL
LIN {X 0,Y 743.922,Z 1055.469,A -85,B 0,C 180,E1 -440.093,E2 -440.093} C_VEL
LIN {X 0,Y 743.921,Z 1062.51,A -85,B 0,C 180,E1 -441.731,E2 -441.731} C_VEL
LIN {X 0,Y 743.898,Z 1068.506,A -85,B 0,C 180,E1 -443.44,E2 -443.44} C_VEL
LIN {X 0,Y 743.916,Z 1073.495,A -85,B 0,C 180,E1 -445.374,E2 -445.374} C_VEL
LIN {X 0,Y 743.912,Z 1076.458,A -85,B 0,C 180,E1 -447.072,E2 -447.072} C_VEL
LIN {X 0,Y 743.91,Z 1078.24,A -85,B 0,C 180,E1 -449.076,E2 -449.076} C_VEL
LIN {X 0,Y 743.894,Z 1078.306,A -85,B 0,C 180,E1 -450.693,E2 -450.693} C_VEL
LIN {X 0,Y 743.906,Z 1077.017,A -85,B 0,C 180,E1 -452.542,E2 -452.542} C_VEL
LIN {X 0,Y 743.901,Z 1073.971,A -85,B 0,C 180,E1 -454.394,E2 -454.394} C_VEL
LIN {X 0,Y 743.913,Z 1070.07,A -85,B 0,C 180,E1 -456.018,E2 -456.018} C_VEL
LIN {X 0,Y 743.916,Z 1063.726,A -85,B 0,C 180,E1 -457.958,E2 -457.958} C_VEL
LIN {X 0,Y 743.917,Z 1056.89,A -85,B 0,C 180,E1 -459.594,E2 -459.594} C_VEL
LIN {X 0,Y 743.973,Z 1047.87,A -85,B 0,C 180,E1 -461.395,E2 -461.395} C_VEL
LIN {X 0,Y 743.998,Z 1037.312,A -85,B 0,C 180,E1 -463.128,E2 -463.128} C_VEL
LIN {X 0,Y 744.045,Z 1026.215,A -85,B 0,C 180,E1 -464.714,E2 -464.714} C_VEL
LIN {X 0,Y 744.124,Z 1012.63,A -85,B 0,C 180,E1 -466.39,E2 -466.39} C_VEL
LIN {X 0,Y 744.184,Z 999.29,A -85,B 0,C 180,E1 -467.839,E2 -467.839} C_VEL
LIN {X 0,Y 744.331,Z 982.32,A -85,B 0,C 180,E1 -469.46,E2 -469.46} C_VEL
LIN {X 0,Y 744.429,Z 966.464,A -85,B 0,C 180,E1 -470.796,E2 -470.796} C_VEL
LIN {X 0,Y 744.599,Z 946.855,A -85,B 0,C 180,E1 -472.252,E2 -472.252} C_VEL
LIN {X 0,Y 744.739,Z 928.436,A -85,B 0,C 180,E1 -473.458,E2 -473.458} C_VEL
LIN {X 0,Y 744.94,Z 906.546,A -85,B 0,C 180,E1 -474.705,E2 -474.705} C_VEL
LIN {X 0,Y 745.09,Z 886.789,A -85,B 0,C 180,E1 -475.687,E2 -475.687} C_VEL
LIN {X 0,Y 745.304,Z 863.327,A -85,B 0,C 180,E1 -476.683,E2 -476.683} C_VEL
LIN {X 0,Y 745.413,Z 843.695,A -85,B 0,C 180,E1 -477.393,E2 -477.393} C_VEL
LIN {X 0,Y 745.617,Z 820.258,A -85,B 0,C 180,E1 -478.104,E2 -478.104} C_VEL
LIN {X 0,Y 745.705,Z 797.579,A -85,B 0,C 180,E1 -478.643,E2 -478.643} C_VEL
LIN {X 0,Y 745.809,Z 777.002,A -85,B 0,C 180,E1 -479.025,E2 -479.025} C_VEL
LIN {X 0,Y 745.904,Z 746.262,A -85,B 0,C 180,E1 -479.418,E2 -479.418} C_VEL
LIN {X 0,Y 746.271,Z 496.111,A -85,B 0,C 180,E1 -482.147,E2 -482.147} C_VEL
LIN {X 0,Y 746.29,Z 379.923,A -85,B 0,C 180,E1 -483.449,E2 -483.449} C_VEL
LIN {X 0,Y 745.547,Z 376.686,A -85,B 0,C 180,E1 -483.542,E2 -483.542} C_VEL
LIN {X 0,Y 745.733,Z 341.211,A -85,B 0,C 180,E1 -485.964,E2 -485.964} C_VEL
LIN {X 0,Y 745.69,Z 333.582,A -85,B 0,C 180,E1 -486.499,E2 -486.499} C_VEL
LIN {X 0,Y 744.038,Z 328.555,A -85,B 0,C 180,E1 -486.969,E2 -486.969} C_VEL
LIN {X 0,Y 743.965,Z 328.554,A -85,B 0,C 180,E1 -489.673,E2 -489.673} C_VEL
LIN {X 0,Y 743.968,Z 328.551,A -85,B 0,C 180,E1 -492.117,E2 -492.117} C_VEL
LIN {X 0,Y 744.04,Z 328.553,A -85,B 0,C 180,E1 -494.981,E2 -494.981} C_VEL
LIN {X 0,Y 743.967,Z 328.552,A -85,B 0,C 180,E1 -497.778,E2 -497.778} C_VEL
LIN {X 0,Y 743.969,Z 328.549,A -85,B 0,C 180,E1 -500.243,E2 -500.243} C_VEL
LIN {X 0,Y 744.038,Z 328.549,A -85,B 0,C 180,E1 -502.983,E2 -502.983} C_VEL
LIN {X 0,Y 743.974,Z 328.552,A -85,B 0,C 180,E1 -505.82,E2 -505.82} C_VEL
LIN {X 0,Y 743.965,Z 328.55,A -85,B 0,C 180,E1 -508.298,E2 -508.298} C_VEL
LIN {X 0,Y 744.039,Z 328.547,A -85,B 0,C 180,E1 -511.028,E2 -511.028} C_VEL
LIN {X 0,Y 743.977,Z 328.553,A -85,B 0,C 180,E1 -513.929,E2 -513.929} C_VEL
LIN {X 0,Y 743.968,Z 328.549,A -85,B 0,C 180,E1 -516.474,E2 -516.474} C_VEL
LIN {X 0,Y 744.036,Z 328.548,A -85,B 0,C 180,E1 -519.22,E2 -519.22} C_VEL
LIN {X 0,Y 743.976,Z 328.552,A -85,B 0,C 180,E1 -522.089,E2 -522.089} C_VEL
LIN {X 0,Y 743.967,Z 328.549,A -85,B 0,C 180,E1 -524.567,E2 -524.567} C_VEL
LIN {X 0,Y 744.04,Z 328.547,A -85,B 0,C 180,E1 -527.329,E2 -527.329} C_VEL
LIN {X 0,Y 743.975,Z 328.553,A -85,B 0,C 180,E1 -530.25,E2 -530.25} C_VEL
LIN {X 0,Y 743.969,Z 328.548,A -85,B 0,C 180,E1 -532.742,E2 -532.742} C_VEL
LIN {X 0,Y 744.037,Z 328.549,A -85,B 0,C 180,E1 -535.53,E2 -535.53} C_VEL
LIN {X 0,Y 743.977,Z 328.552,A -85,B 0,C 180,E1 -538.383,E2 -538.383} C_VEL
LIN {X 0,Y 743.972,Z 328.549,A -85,B 0,C 180,E1 -540.924,E2 -540.924} C_VEL
LIN {X 0,Y 744.039,Z 328.548,A -85,B 0,C 180,E1 -543.698,E2 -543.698} C_VEL
LIN {X 0,Y 743.976,Z 328.55,A -85,B 0,C 180,E1 -546.56,E2 -546.56} C_VEL
LIN {X 0,Y 744.029,Z 328.555,A -85,B 0,C 180,E1 -548.121,E2 -548.121} C_VEL
LIN {X 0,Y 742.978,Z 328.677,A -85,B 0,C 180,E1 -548.714,E2 -548.714} C_VEL
LIN {X 0,Y 736.559,Z 329.481,A -85,B 0,C 180,E1 -550.376,E2 -550.376} C_VEL
LIN {X 0,Y 736.03,Z 329.538,A -85,B 0,C 180,E1 -550.807,E2 -550.807} C_VEL
LIN {X 0,Y 736.059,Z 329.537,A -85,B 0,C 180,E1 -553.434,E2 -553.434} C_VEL
LIN {X 0,Y 736.058,Z 329.542,A -85,B 0,C 180,E1 -556.494,E2 -556.494} C_VEL
LIN {X 0,Y 736.031,Z 329.538,A -85,B 0,C 180,E1 -559.111,E2 -559.111} C_VEL
LIN {X 0,Y 736.094,Z 329.535,A -85,B 0,C 180,E1 -561.851,E2 -561.851} C_VEL
LIN {X 0,Y 736.042,Z 329.542,A -85,B 0,C 180,E1 -564.82,E2 -564.82} C_VEL
LIN {X 0,Y 736.038,Z 329.537,A -85,B 0,C 180,E1 -567.421,E2 -567.421} C_VEL
LIN {X 0,Y 736.099,Z 329.54,A -85,B 0,C 180,E1 -570.262,E2 -570.262} C_VEL
LIN {X 0,Y 736.035,Z 329.541,A -85,B 0,C 180,E1 -573.101,E2 -573.101} C_VEL
LIN {X 0,Y 736.052,Z 329.537,A -85,B 0,C 180,E1 -575.742,E2 -575.742} C_VEL
LIN {X 0,Y 736.074,Z 329.544,A -85,B 0,C 180,E1 -578.773,E2 -578.773} C_VEL
LIN {X 0,Y 736.032,Z 329.54,A -85,B 0,C 180,E1 -581.421,E2 -581.421} C_VEL
LIN {X 0,Y 736.093,Z 329.535,A -85,B 0,C 180,E1 -584.175,E2 -584.175} C_VEL
LIN {X 0,Y 736.05,Z 329.544,A -85,B 0,C 180,E1 -587.111,E2 -587.111} C_VEL
LIN {X 0,Y 736.036,Z 329.54,A -85,B 0,C 180,E1 -589.712,E2 -589.712} C_VEL
LIN {X 0,Y 736.1,Z 329.54,A -85,B 0,C 180,E1 -592.516,E2 -592.516} C_VEL
LIN {X 0,Y 736.114,Z 329.662,A -85,B 0,C 180,E1 -594.708,E2 -594.708} C_VEL
LIN {X 0,Y 738.341,Z 337.037,A -85,B 0,C 180,E1 -595.382,E2 -595.382} C_VEL
LIN {X 0,Y 738.386,Z 347.916,A -85,B 0,C 180,E1 -596.167,E2 -596.167} C_VEL
LIN {X 0,Y 739.745,Z 353.952,A -85,B 0,C 180,E1 -596.306,E2 -596.306} C_VEL
LIN {X 0,Y 739.208,Z 592.54,A -85,B 0,C 180,E1 -598.969,E2 -598.969} C_VEL
LIN {X 0,Y 738.868,Z 736.609,A -85,B 0,C 180,E1 -600.564,E2 -600.564} C_VEL
LIN {X 0,Y 738.666,Z 761.866,A -85,B 0,C 180,E1 -600.981,E2 -600.981} C_VEL
LIN {X 0,Y 738.511,Z 783.407,A -85,B 0,C 180,E1 -601.471,E2 -601.471} C_VEL
LIN {X 0,Y 738.319,Z 806.587,A -85,B 0,C 180,E1 -602.124,E2 -602.124} C_VEL
LIN {X 0,Y 738.047,Z 829.322,A -85,B 0,C 180,E1 -602.922,E2 -602.922} C_VEL
LIN {X 0,Y 737.828,Z 850.242,A -85,B 0,C 180,E1 -603.784,E2 -603.784} C_VEL
LIN {X 0,Y 737.503,Z 873.1,A -85,B 0,C 180,E1 -604.89,E2 -604.89} C_VEL
LIN {X 0,Y 737.281,Z 892.843,A -85,B 0,C 180,E1 -605.993,E2 -605.993} C_VEL
LIN {X 0,Y 736.988,Z 913.797,A -85,B 0,C 180,E1 -607.337,E2 -607.337} C_VEL
LIN {X 0,Y 736.78,Z 932.635,A -85,B 0,C 180,E1 -608.712,E2 -608.712} C_VEL
LIN {X 0,Y 736.546,Z 950.207,A -85,B 0,C 180,E1 -610.183,E2 -610.183} C_VEL
LIN {X 0,Y 736.394,Z 966.535,A -85,B 0,C 180,E1 -611.72,E2 -611.72} C_VEL
LIN {X 0,Y 736.242,Z 981.533,A -85,B 0,C 180,E1 -613.348,E2 -613.348} C_VEL
LIN {X 0,Y 736.124,Z 995.314,A -85,B 0,C 180,E1 -615.044,E2 -615.044} C_VEL
LIN {X 0,Y 736.045,Z 1007.021,A -85,B 0,C 180,E1 -616.728,E2 -616.728} C_VEL
LIN {X 0,Y 735.997,Z 1017.61,A -85,B 0,C 180,E1 -618.48,E2 -618.48} C_VEL
LIN {X 0,Y 735.93,Z 1026.689,A -85,B 0,C 180,E1 -620.301,E2 -620.301} C_VEL
LIN {X 0,Y 735.938,Z 1033.248,A -85,B 0,C 180,E1 -621.877,E2 -621.877} C_VEL
LIN {X 0,Y 735.92,Z 1039.746,A -85,B 0,C 180,E1 -623.838,E2 -623.838} C_VEL
LIN {X 0,Y 735.915,Z 1043.88,A -85,B 0,C 180,E1 -625.558,E2 -625.558} C_VEL
LIN {X 0,Y 735.893,Z 1046.844,A -85,B 0,C 180,E1 -627.352,E2 -627.352} C_VEL
LIN {X 0,Y 735.899,Z 1048.271,A -85,B 0,C 180,E1 -629.222,E2 -629.222} C_VEL
LIN {X 0,Y 735.904,Z 1048.275,A -85,B 0,C 180,E1 -630.856,E2 -630.856} C_VEL
LIN {X 0,Y 735.9,Z 1046.749,A -85,B 0,C 180,E1 -632.804,E2 -632.804} C_VEL
LIN {X 0,Y 735.914,Z 1043.904,A -85,B 0,C 180,E1 -634.52,E2 -634.52} C_VEL
LIN {X 0,Y 735.914,Z 1039.776,A -85,B 0,C 180,E1 -636.24,E2 -636.24} C_VEL
LIN {X 0,Y 735.931,Z 1033.292,A -85,B 0,C 180,E1 -638.202,E2 -638.202} C_VEL
LIN {X 0,Y 735.935,Z 1026.738,A -85,B 0,C 180,E1 -639.778,E2 -639.778} C_VEL
LIN {X 0,Y 735.997,Z 1017.67,A -85,B 0,C 180,E1 -641.599,E2 -641.599} C_VEL
LIN {X 0,Y 736.045,Z 1007.085,A -85,B 0,C 180,E1 -643.352,E2 -643.352} C_VEL
LIN {X 0,Y 736.125,Z 995.38,A -85,B 0,C 180,E1 -645.037,E2 -645.037} C_VEL
LIN {X 0,Y 736.246,Z 981.608,A -85,B 0,C 180,E1 -646.733,E2 -646.733} C_VEL
LIN {X 0,Y 736.393,Z 966.671,A -85,B 0,C 180,E1 -648.355,E2 -648.355} C_VEL
LIN {X 0,Y 736.541,Z 950.966,A -85,B 0,C 180,E1 -649.84,E2 -649.84} C_VEL
LIN {X 0,Y 736.768,Z 933.793,A -85,B 0,C 180,E1 -651.288,E2 -651.288} C_VEL
LIN {X 0,Y 736.979,Z 915.086,A -85,B 0,C 180,E1 -652.663,E2 -652.663} C_VEL
LIN {X 0,Y 737.27,Z 895.054,A -85,B 0,C 180,E1 -653.969,E2 -653.969} C_VEL
LIN {X 0,Y 737.497,Z 873.98,A -85,B 0,C 180,E1 -655.153,E2 -655.153} C_VEL
LIN {X 0,Y 737.816,Z 852.259,A -85,B 0,C 180,E1 -656.219,E2 -656.219} C_VEL
LIN {X 0,Y 738.042,Z 830.058,A -85,B 0,C 180,E1 -657.14,E2 -657.14} C_VEL
LIN {X 0,Y 738.307,Z 807.324,A -85,B 0,C 180,E1 -657.943,E2 -657.943} C_VEL
LIN {X 0,Y 738.511,Z 783.714,A -85,B 0,C 180,E1 -658.611,E2 -658.611} C_VEL
LIN {X 0,Y 738.669,Z 762.407,A -85,B 0,C 180,E1 -659.097,E2 -659.097} C_VEL
LIN {X 0,Y 738.868,Z 736.968,A -85,B 0,C 180,E1 -659.521,E2 -659.521} C_VEL
LIN {X 0,Y 739.113,Z 633.855,A -85,B 0,C 180,E1 -660.668,E2 -660.668} C_VEL
LIN {X 0,Y 739.652,Z 387.908,A -85,B 0,C 180,E1 -663.401,E2 -663.401} C_VEL
LIN {X 0,Y 739.573,Z 352.393,A -85,B 0,C 180,E1 -663.81,E2 -663.81} C_VEL
LIN {X 0,Y 738.297,Z 347.097,A -85,B 0,C 180,E1 -663.963,E2 -663.963} C_VEL
LIN {X 0,Y 738.25,Z 336.343,A -85,B 0,C 180,E1 -664.765,E2 -664.765} C_VEL
LIN {X 0,Y 736.1,Z 329.543,A -85,B 0,C 180,E1 -665.411,E2 -665.411} C_VEL
LIN {X 0,Y 736.03,Z 329.542,A -85,B 0,C 180,E1 -668.278,E2 -668.278} C_VEL
LIN {X 0,Y 736.039,Z 329.544,A -85,B 0,C 180,E1 -670.828,E2 -670.828} C_VEL
LIN {X 0,Y 736.095,Z 329.532,A -85,B 0,C 180,E1 -673.742,E2 -673.742} C_VEL
LIN {X 0,Y 736.026,Z 329.541,A -85,B 0,C 180,E1 -676.505,E2 -676.505} C_VEL
LIN {X 0,Y 736.051,Z 329.537,A -85,B 0,C 180,E1 -679.097,E2 -679.097} C_VEL
LIN {X 0,Y 736.05,Z 329.537,A -85,B 0,C 180,E1 -682.217,E2 -682.217} C_VEL
LIN {X 0,Y 736.026,Z 329.541,A -85,B 0,C 180,E1 -684.735,E2 -684.735} C_VEL
LIN {X 0,Y 736.067,Z 329.543,A -85,B 0,C 180,E1 -687.376,E2 -687.376} C_VEL
LIN {X 0,Y 736.047,Z 329.538,A -85,B 0,C 180,E1 -690.391,E2 -690.391} C_VEL
LIN {X 0,Y 736.025,Z 329.539,A -85,B 0,C 180,E1 -692.929,E2 -692.929} C_VEL
LIN {X 0,Y 736.082,Z 329.544,A -85,B 0,C 180,E1 -695.609,E2 -695.609} C_VEL
LIN {X 0,Y 736.042,Z 329.538,A -85,B 0,C 180,E1 -698.566,E2 -698.566} C_VEL
LIN {X 0,Y 736.025,Z 329.539,A -85,B 0,C 180,E1 -701.054,E2 -701.054} C_VEL
LIN {X 0,Y 736.082,Z 329.544,A -85,B 0,C 180,E1 -703.75,E2 -703.75} C_VEL
LIN {X 0,Y 736.041,Z 329.538,A -85,B 0,C 180,E1 -706.727,E2 -706.727} C_VEL
LIN {X 0,Y 736.026,Z 329.538,A -85,B 0,C 180,E1 -709.274,E2 -709.274} C_VEL
LIN {X 0,Y 736.098,Z 329.543,A -85,B 0,C 180,E1 -712.036,E2 -712.036} C_VEL
LIN {X 0,Y 736.035,Z 329.538,A -85,B 0,C 180,E1 -714.934,E2 -714.934} C_VEL
LIN {X 0,Y 736.027,Z 329.541,A -85,B 0,C 180,E1 -717.431,E2 -717.431} C_VEL
LIN {X 0,Y 736.102,Z 329.542,A -85,B 0,C 180,E1 -720.233,E2 -720.233} C_VEL
LIN {X 0,Y 736.031,Z 329.536,A -85,B 0,C 180,E1 -723.115,E2 -723.115} C_VEL
LIN {X 0,Y 736.028,Z 329.541,A -85,B 0,C 180,E1 -725.613,E2 -725.613} C_VEL
LIN {X 0,Y 736.1,Z 329.54,A -85,B 0,C 180,E1 -728.436,E2 -728.436} C_VEL
LIN {X 0,Y 736.03,Z 329.538,A -85,B 0,C 180,E1 -731.281,E2 -731.281} C_VEL
LIN {X 0,Y 736.028,Z 329.541,A -85,B 0,C 180,E1 -733.754,E2 -733.754} C_VEL
LIN {X 0,Y 736.1,Z 329.539,A -85,B 0,C 180,E1 -736.574,E2 -736.574} C_VEL
LIN {X 0,Y 736.032,Z 329.538,A -85,B 0,C 180,E1 -739.358,E2 -739.358} C_VEL
LIN {X 0,Y 736.027,Z 329.54,A -85,B 0,C 180,E1 -741.853,E2 -741.853} C_VEL
LIN {X 0,Y 736.101,Z 329.542,A -85,B 0,C 180,E1 -744.647,E2 -744.647} C_VEL
LIN {X 0,Y 736.031,Z 329.538,A -85,B 0,C 180,E1 -747.509,E2 -747.509} C_VEL
LIN {X 0,Y 736.027,Z 329.542,A -85,B 0,C 180,E1 -749.995,E2 -749.995} C_VEL
LIN {X 0,Y 736.1,Z 329.542,A -85,B 0,C 180,E1 -752.773,E2 -752.773} C_VEL
LIN {X 0,Y 736.032,Z 329.54,A -85,B 0,C 180,E1 -755.647,E2 -755.647} C_VEL
LIN {X 0,Y 736.029,Z 329.542,A -85,B 0,C 180,E1 -758.179,E2 -758.179} C_VEL
LIN {X 0,Y 736.099,Z 329.537,A -85,B 0,C 180,E1 -761.071,E2 -761.071} C_VEL
LIN {X 0,Y 736.028,Z 329.539,A -85,B 0,C 180,E1 -763.855,E2 -763.855} C_VEL
LIN {X 0,Y 736.031,Z 329.542,A -85,B 0,C 180,E1 -766.361,E2 -766.361} C_VEL
LIN {X 0,Y 736.094,Z 329.541,A -85,B 0,C 180,E1 -769.286,E2 -769.286} C_VEL
LIN {X 0,Y 736.027,Z 329.545,A -85,B 0,C 180,E1 -772.019,E2 -772.019} C_VEL
LIN {X 0,Y 736.059,Z 329.629,A -85,B 0,C 180,E1 -772.661,E2 -772.661} C_VEL
LIN {X 0,Y 738.755,Z 337.511,A -85,B 0,C 180,E1 -773.381,E2 -773.381} C_VEL
LIN {X 0,Y 738.447,Z 373.272,A -85,B 0,C 180,E1 -775.858,E2 -775.858} C_VEL
LIN {X 0,Y 738.5,Z 377.445,A -85,B 0,C 180,E1 -776.122,E2 -776.122} C_VEL
LIN {X 0,Y 739.784,Z 383.419,A -85,B 0,C 180,E1 -776.257,E2 -776.257} C_VEL
LIN {X 0,Y 739.163,Z 641.592,A -85,B 0,C 180,E1 -779.133,E2 -779.133} C_VEL
LIN {X 0,Y 738.866,Z 766.74,A -85,B 0,C 180,E1 -780.521,E2 -780.521} C_VEL
LIN {X 0,Y 738.666,Z 792.02,A -85,B 0,C 180,E1 -780.939,E2 -780.939} C_VEL
LIN {X 0,Y 738.511,Z 813.466,A -85,B 0,C 180,E1 -781.427,E2 -781.427} C_VEL
LIN {X 0,Y 738.321,Z 836.618,A -85,B 0,C 180,E1 -782.08,E2 -782.08} C_VEL
LIN {X 0,Y 738.045,Z 859.541,A -85,B 0,C 180,E1 -782.885,E2 -782.885} C_VEL
LIN {X 0,Y 737.827,Z 880.232,A -85,B 0,C 180,E1 -783.739,E2 -783.739} C_VEL
LIN {X 0,Y 737.503,Z 903.139,A -85,B 0,C 180,E1 -784.847,E2 -784.847} C_VEL
LIN {X 0,Y 737.28,Z 922.885,A -85,B 0,C 180,E1 -785.95,E2 -785.95} C_VEL
LIN {X 0,Y 736.992,Z 943.233,A -85,B 0,C 180,E1 -787.253,E2 -787.253} C_VEL
LIN {X 0,Y 736.792,Z 961.105,A -85,B 0,C 180,E1 -788.551,E2 -788.551} C_VEL
LIN {X 0,Y 736.567,Z 978.603,A -85,B 0,C 180,E1 -789.996,E2 -789.996} C_VEL
LIN {X 0,Y 736.424,Z 994.493,A -85,B 0,C 180,E1 -791.475,E2 -791.475} C_VEL
LIN {X 0,Y 736.245,Z 1009.801,A -85,B 0,C 180,E1 -793.104,E2 -793.104} C_VEL
LIN {X 0,Y 736.159,Z 1022.668,A -85,B 0,C 180,E1 -794.658,E2 -794.658} C_VEL
LIN {X 0,Y 736.056,Z 1035.753,A -85,B 0,C 180,E1 -796.488,E2 -796.488} C_VEL
LIN {X 0,Y 735.988,Z 1045.128,A -85,B 0,C 180,E1 -798.007,E2 -798.007} C_VEL
LIN {X 0,Y 735.962,Z 1054.76,A -85,B 0,C 180,E1 -799.827,E2 -799.827} C_VEL
LIN {X 0,Y 735.918,Z 1062.206,A -85,B 0,C 180,E1 -801.562,E2 -801.562} C_VEL
LIN {X 0,Y 735.911,Z 1067.997,A -85,B 0,C 180,E1 -803.211,E2 -803.211} C_VEL
LIN {X 0,Y 735.917,Z 1073.178,A -85,B 0,C 180,E1 -805.168,E2 -805.168} C_VEL
LIN {X 0,Y 735.916,Z 1076.234,A -85,B 0,C 180,E1 -806.884,E2 -806.884} C_VEL
LIN {X 0,Y 735.907,Z 1078.149,A -85,B 0,C 180,E1 -808.754,E2 -808.754} C_VEL
LIN {X 0,Y 735.891,Z 1078.351,A -85,B 0,C 180,E1 -810.545,E2 -810.545} C_VEL
LIN {X 0,Y 735.914,Z 1077.297,A -85,B 0,C 180,E1 -812.258,E2 -812.258} C_VEL
LIN {X 0,Y 735.908,Z 1074.445,A -85,B 0,C 180,E1 -814.208,E2 -814.208} C_VEL
LIN {X 0,Y 735.917,Z 1070.688,A -85,B 0,C 180,E1 -815.849,E2 -815.849} C_VEL
LIN {X 0,Y 735.911,Z 1064.936,A -85,B 0,C 180,E1 -817.73,E2 -817.73} C_VEL
LIN {X 0,Y 735.931,Z 1057.601,A -85,B 0,C 180,E1 -819.541,E2 -819.541} C_VEL
LIN {X 0,Y 735.974,Z 1049.927,A -85,B 0,C 180,E1 -821.123,E2 -821.123} C_VEL
LIN {X 0,Y 736.039,Z 1038.526,A -85,B 0,C 180,E1 -823.086,E2 -823.086} C_VEL
LIN {X 0,Y 736.104,Z 1027.954,A -85,B 0,C 180,E1 -824.635,E2 -824.635} C_VEL
LIN {X 0,Y 736.23,Z 1014.046,A -85,B 0,C 180,E1 -826.409,E2 -826.409} C_VEL
LIN {X 0,Y 736.33,Z 1000.069,A -85,B 0,C 180,E1 -827.954,E2 -827.954} C_VEL
LIN {X 0,Y 736.542,Z 983.248,A -85,B 0,C 180,E1 -829.592,E2 -829.592} C_VEL
LIN {X 0,Y 736.708,Z 966.807,A -85,B 0,C 180,E1 -830.996,E2 -830.996} C_VEL
LIN {X 0,Y 736.965,Z 946.857,A -85,B 0,C 180,E1 -832.495,E2 -832.495} C_VEL
LIN {X 0,Y 737.195,Z 928.356,A -85,B 0,C 180,E1 -833.718,E2 -833.718} C_VEL
LIN {X 0,Y 737.479,Z 906.348,A -85,B 0,C 180,E1 -834.982,E2 -834.982} C_VEL
LIN {X 0,Y 737.72,Z 886.791,A -85,B 0,C 180,E1 -835.963,E2 -835.963} C_VEL
LIN {X 0,Y 738.022,Z 863.386,A -85,B 0,C 180,E1 -836.966,E2 -836.966} C_VEL
LIN {X 0,Y 738.198,Z 843.699,A -85,B 0,C 180,E1 -837.684,E2 -837.684} C_VEL
LIN {X 0,Y 738.494,Z 820.046,A -85,B 0,C 180,E1 -838.405,E2 -838.405} C_VEL
LIN {X 0,Y 738.641,Z 797.322,A -85,B 0,C 180,E1 -838.949,E2 -838.949} C_VEL
LIN {X 0,Y 738.792,Z 776.078,A -85,B 0,C 180,E1 -839.344,E2 -839.344} C_VEL
LIN {X 0,Y 738.933,Z 744.926,A -85,B 0,C 180,E1 -839.738,E2 -839.738} C_VEL
LIN {X 0,Y 739.501,Z 493.624,A -85,B 0,C 180,E1 -842.505,E2 -842.505} C_VEL
LIN {X 0,Y 739.604,Z 381.804,A -85,B 0,C 180,E1 -843.771,E2 -843.771} C_VEL
LIN {X 0,Y 738.409,Z 376.686,A -85,B 0,C 180,E1 -843.91,E2 -843.91} C_VEL
LIN {X 0,Y 738.712,Z 341.299,A -85,B 0,C 180,E1 -846.354,E2 -846.354} C_VEL
LIN {X 0,Y 738.481,Z 336.304,A -85,B 0,C 180,E1 -846.72,E2 -846.72} C_VEL
LIN {X 0,Y 736.044,Z 329.548,A -85,B 0,C 180,E1 -847.372,E2 -847.372} C_VEL
LIN {X 0,Y 736.024,Z 329.543,A -85,B 0,C 180,E1 -849.882,E2 -849.882} C_VEL
LIN {X 0,Y 736.063,Z 329.538,A -85,B 0,C 180,E1 -852.47,E2 -852.47} C_VEL
LIN {X 0,Y 736.048,Z 329.543,A -85,B 0,C 180,E1 -855.495,E2 -855.495} C_VEL
LIN {X 0,Y 736.025,Z 329.54,A -85,B 0,C 180,E1 -858.057,E2 -858.057} C_VEL
LIN {X 0,Y 736.082,Z 329.536,A -85,B 0,C 180,E1 -860.74,E2 -860.74} C_VEL
LIN {X 0,Y 736.043,Z 329.534,A -85,B 0,C 180,E1 -863.68,E2 -863.68} C_VEL
LIN {X 0,Y 736.027,Z 329.538,A -85,B 0,C 180,E1 -866.246,E2 -866.246} C_VEL
LIN {X 0,Y 736.099,Z 329.535,A -85,B 0,C 180,E1 -869.014,E2 -869.014} C_VEL
LIN {X 0,Y 736.039,Z 329.54,A -85,B 0,C 180,E1 -871.875,E2 -871.875} C_VEL
LIN {X 0,Y 736.03,Z 329.539,A -85,B 0,C 180,E1 -874.427,E2 -874.427} C_VEL
LIN {X 0,Y 736.101,Z 329.537,A -85,B 0,C 180,E1 -877.224,E2 -877.224} C_VEL
LIN {X 0,Y 736.036,Z 329.541,A -85,B 0,C 180,E1 -880.063,E2 -880.063} C_VEL
LIN {X 0,Y 736.032,Z 329.539,A -85,B 0,C 180,E1 -882.61,E2 -882.61} C_VEL
LIN {X 0,Y 736.098,Z 329.538,A -85,B 0,C 180,E1 -885.446,E2 -885.446} C_VEL
LIN {X 0,Y 736.035,Z 329.54,A -85,B 0,C 180,E1 -888.242,E2 -888.242} C_VEL
LIN {X 0,Y 736.033,Z 329.539,A -85,B 0,C 180,E1 -890.776,E2 -890.776} C_VEL
LIN {X 0,Y 736.099,Z 329.537,A -85,B 0,C 180,E1 -893.605,E2 -893.605} C_VEL
LIN {X 0,Y 736.034,Z 329.539,A -85,B 0,C 180,E1 -896.417,E2 -896.417} C_VEL
LIN {X 0,Y 736.038,Z 329.538,A -85,B 0,C 180,E1 -898.988,E2 -898.988} C_VEL
LIN {X 0,Y 736.095,Z 329.542,A -85,B 0,C 180,E1 -901.946,E2 -901.946} C_VEL
LIN {X 0,Y 736.03,Z 329.54,A -85,B 0,C 180,E1 -904.675,E2 -904.675} C_VEL
LIN {X 0,Y 736.05,Z 329.535,A -85,B 0,C 180,E1 -907.258,E2 -907.258} C_VEL
LIN {X 0,Y 736.065,Z 329.541,A -85,B 0,C 180,E1 -910.33,E2 -910.33} C_VEL
LIN {X 0,Y 736.03,Z 329.538,A -85,B 0,C 180,E1 -910.807,E2 -910.807} C_VEL
LIN {X 0,Y 735.031,Z 329.666,A -85,B 0,C 180,E1 -911.407,E2 -911.407} C_VEL
LIN {X 0,Y 728.618,Z 330.465,A -85,B 0,C 180,E1 -913.086,E2 -913.086} C_VEL
LIN {X 0,Y 728.13,Z 330.525,A -85,B 0,C 180,E1 -913.523,E2 -913.523} C_VEL
LIN {X 0,Y 728.113,Z 330.531,A -85,B 0,C 180,E1 -916.557,E2 -916.557} C_VEL
LIN {X 0,Y 728.094,Z 330.527,A -85,B 0,C 180,E1 -919.161,E2 -919.161} C_VEL
LIN {X 0,Y 728.16,Z 330.525,A -85,B 0,C 180,E1 -921.932,E2 -921.932} C_VEL
LIN {X 0,Y 728.101,Z 330.53,A -85,B 0,C 180,E1 -924.849,E2 -924.849} C_VEL
LIN {X 0,Y 728.104,Z 330.525,A -85,B 0,C 180,E1 -927.479,E2 -927.479} C_VEL
LIN {X 0,Y 728.16,Z 330.531,A -85,B 0,C 180,E1 -930.445,E2 -930.445} C_VEL
LIN {X 0,Y 728.094,Z 330.529,A -85,B 0,C 180,E1 -933.245,E2 -933.245} C_VEL
LIN {X 0,Y 728.145,Z 330.524,A -85,B 0,C 180,E1 -935.996,E2 -935.996} C_VEL
LIN {X 0,Y 728.111,Z 330.531,A -85,B 0,C 180,E1 -938.989,E2 -938.989} C_VEL
LIN {X 0,Y 728.096,Z 330.529,A -85,B 0,C 180,E1 -941.552,E2 -941.552} C_VEL
LIN {X 0,Y 728.16,Z 330.529,A -85,B 0,C 180,E1 -944.435,E2 -944.435} C_VEL
LIN {X 0,Y 728.101,Z 330.532,A -85,B 0,C 180,E1 -947.283,E2 -947.283} C_VEL
LIN {X 0,Y 728.109,Z 330.529,A -85,B 0,C 180,E1 -949.905,E2 -949.905} C_VEL
LIN {X 0,Y 728.148,Z 330.527,A -85,B 0,C 180,E1 -952.927,E2 -952.927} C_VEL
LIN {X 0,Y 728.16,Z 330.619,A -85,B 0,C 180,E1 -954.336,E2 -954.336} C_VEL
LIN {X 0,Y 731.181,Z 340.204,A -85,B 0,C 180,E1 -955.233,E2 -955.233} C_VEL
LIN {X 0,Y 731.241,Z 347.971,A -85,B 0,C 180,E1 -955.791,E2 -955.791} C_VEL
LIN {X 0,Y 733.078,Z 355.782,A -85,B 0,C 180,E1 -955.979,E2 -955.979} C_VEL
LIN {X 0,Y 732.345,Z 594.754,A -85,B 0,C 180,E1 -958.669,E2 -958.669} C_VEL
LIN {X 0,Y 731.892,Z 736.76,A -85,B 0,C 180,E1 -960.257,E2 -960.257} C_VEL
LIN {X 0,Y 731.632,Z 762.195,A -85,B 0,C 180,E1 -960.682,E2 -960.682} C_VEL
LIN {X 0,Y 731.418,Z 783.786,A -85,B 0,C 180,E1 -961.177,E2 -961.177} C_VEL
LIN {X 0,Y 731.151,Z 807.276,A -85,B 0,C 180,E1 -961.848,E2 -961.848} C_VEL
LIN {X 0,Y 730.795,Z 829.341,A -85,B 0,C 180,E1 -962.631,E2 -962.631} C_VEL
LIN {X 0,Y 730.492,Z 851.009,A -85,B 0,C 180,E1 -963.533,E2 -963.533} C_VEL
LIN {X 0,Y 730.066,Z 873.543,A -85,B 0,C 180,E1 -964.639,E2 -964.639} C_VEL
LIN {X 0,Y 729.756,Z 893.582,A -85,B 0,C 180,E1 -965.772,E2 -965.772} C_VEL
LIN {X 0,Y 729.377,Z 914.098,A -85,B 0,C 180,E1 -967.108,E2 -967.108} C_VEL
LIN {X 0,Y 729.084,Z 933.218,A -85,B 0,C 180,E1 -968.52,E2 -968.52} C_VEL
LIN {X 0,Y 728.771,Z 950.905,A -85,B 0,C 180,E1 -970.025,E2 -970.025} C_VEL
LIN {X 0,Y 728.558,Z 967.318,A -85,B 0,C 180,E1 -971.6,E2 -971.6} C_VEL
LIN {X 0,Y 728.355,Z 981.539,A -85,B 0,C 180,E1 -973.162,E2 -973.162} C_VEL
LIN {X 0,Y 728.209,Z 995.319,A -85,B 0,C 180,E1 -974.877,E2 -974.877} C_VEL
LIN {X 0,Y 728.094,Z 1007.026,A -85,B 0,C 180,E1 -976.58,E2 -976.58} C_VEL
LIN {X 0,Y 728.023,Z 1017.612,A -85,B 0,C 180,E1 -978.352,E2 -978.352} C_VEL
LIN {X 0,Y 727.945,Z 1026.691,A -85,B 0,C 180,E1 -980.193,E2 -980.193} C_VEL
LIN {X 0,Y 727.94,Z 1033.25,A -85,B 0,C 180,E1 -981.787,E2 -981.787} C_VEL
LIN {X 0,Y 727.919,Z 1039.747,A -85,B 0,C 180,E1 -983.77,E2 -983.77} C_VEL
LIN {X 0,Y 727.916,Z 1043.881,A -85,B 0,C 180,E1 -985.509,E2 -985.509} C_VEL
LIN {X 0,Y 727.893,Z 1046.845,A -85,B 0,C 180,E1 -987.323,E2 -987.323} C_VEL
LIN {X 0,Y 727.899,Z 1048.271,A -85,B 0,C 180,E1 -989.213,E2 -989.213} C_VEL
LIN {X 0,Y 727.905,Z 1048.275,A -85,B 0,C 180,E1 -990.866,E2 -990.866} C_VEL
LIN {X 0,Y 727.902,Z 1046.748,A -85,B 0,C 180,E1 -992.835,E2 -992.835} C_VEL
LIN {X 0,Y 727.916,Z 1043.903,A -85,B 0,C 180,E1 -994.57,E2 -994.57} C_VEL
LIN {X 0,Y 727.913,Z 1039.775,A -85,B 0,C 180,E1 -996.309,E2 -996.309} C_VEL
LIN {X 0,Y 727.935,Z 1033.29,A -85,B 0,C 180,E1 -998.293,E2 -998.293} C_VEL
LIN {X 0,Y 727.95,Z 1026.736,A -85,B 0,C 180,E1 -999.887,E2 -999.887} C_VEL
LIN {X 0,Y 728.024,Z 1017.666,A -85,B 0,C 180,E1 -1001.728,E2 -1001.728} C_VEL
LIN {X 0,Y 728.09,Z 1007.083,A -85,B 0,C 180,E1 -1003.501,E2 -1003.501} C_VEL
LIN {X 0,Y 728.209,Z 995.378,A -85,B 0,C 180,E1 -1005.204,E2 -1005.204} C_VEL
LIN {X 0,Y 728.356,Z 981.605,A -85,B 0,C 180,E1 -1006.92,E2 -1006.92} C_VEL
LIN {X 0,Y 728.578,Z 966.606,A -85,B 0,C 180,E1 -1008.566,E2 -1008.566} C_VEL
LIN {X 0,Y 728.783,Z 950.031,A -85,B 0,C 180,E1 -1010.144,E2 -1010.144} C_VEL
LIN {X 0,Y 729.088,Z 932.94,A -85,B 0,C 180,E1 -1011.591,E2 -1011.591} C_VEL
LIN {X 0,Y 729.371,Z 914.301,A -85,B 0,C 180,E1 -1012.968,E2 -1012.968} C_VEL
LIN {X 0,Y 729.75,Z 894.375,A -85,B 0,C 180,E1 -1014.271,E2 -1014.271} C_VEL
LIN {X 0,Y 730.058,Z 873.974,A -85,B 0,C 180,E1 -1015.428,E2 -1015.428} C_VEL
LIN {X 0,Y 730.481,Z 852.251,A -85,B 0,C 180,E1 -1016.502,E2 -1016.502} C_VEL
LIN {X 0,Y 730.781,Z 830.499,A -85,B 0,C 180,E1 -1017.414,E2 -1017.414} C_VEL
LIN {X 0,Y 731.115,Z 808.589,A -85,B 0,C 180,E1 -1018.198,E2 -1018.198} C_VEL
LIN {X 0,Y 731.417,Z 784.45,A -85,B 0,C 180,E1 -1018.895,E2 -1018.895} C_VEL
LIN {X 0,Y 731.627,Z 763.291,A -85,B 0,C 180,E1 -1019.385,E2 -1019.385} C_VEL
LIN {X 0,Y 731.89,Z 737.428,A -85,B 0,C 180,E1 -1019.824,E2 -1019.824} C_VEL
LIN {X 0,Y 732.169,Z 653.483,A -85,B 0,C 180,E1 -1020.77,E2 -1020.77} C_VEL
LIN {X 0,Y 732.915,Z 405.17,A -85,B 0,C 180,E1 -1023.549,E2 -1023.549} C_VEL
LIN {X 0,Y 732.874,Z 354.046,A -85,B 0,C 180,E1 -1024.142,E2 -1024.142} C_VEL
LIN {X 0,Y 731.138,Z 347.373,A -85,B 0,C 180,E1 -1024.32,E2 -1024.32} C_VEL
LIN {X 0,Y 731.089,Z 339.404,A -85,B 0,C 180,E1 -1024.923,E2 -1024.923} C_VEL
LIN {X 0,Y 728.132,Z 330.533,A -85,B 0,C 180,E1 -1025.78,E2 -1025.78} C_VEL
LIN {X 0,Y 728.087,Z 330.533,A -85,B 0,C 180,E1 -1028.483,E2 -1028.483} C_VEL
LIN {X 0,Y 728.149,Z 330.532,A -85,B 0,C 180,E1 -1031.234,E2 -1031.234} C_VEL
LIN {X 0,Y 728.1,Z 330.522,A -85,B 0,C 180,E1 -1034.204,E2 -1034.204} C_VEL
LIN {X 0,Y 728.09,Z 330.532,A -85,B 0,C 180,E1 -1036.742,E2 -1036.742} C_VEL
LIN {X 0,Y 728.161,Z 330.527,A -85,B 0,C 180,E1 -1039.598,E2 -1039.598} C_VEL
LIN {X 0,Y 728.094,Z 330.527,A -85,B 0,C 180,E1 -1042.429,E2 -1042.429} C_VEL
LIN {X 0,Y 728.093,Z 330.531,A -85,B 0,C 180,E1 -1044.967,E2 -1044.967} C_VEL
LIN {X 0,Y 728.16,Z 330.527,A -85,B 0,C 180,E1 -1047.806,E2 -1047.806} C_VEL
LIN {X 0,Y 728.091,Z 330.529,A -85,B 0,C 180,E1 -1050.642,E2 -1050.642} C_VEL
LIN {X 0,Y 728.094,Z 330.528,A -85,B 0,C 180,E1 -1053.14,E2 -1053.14} C_VEL
LIN {X 0,Y 728.161,Z 330.525,A -85,B 0,C 180,E1 -1056.017,E2 -1056.017} C_VEL
LIN {X 0,Y 728.088,Z 330.529,A -85,B 0,C 180,E1 -1058.827,E2 -1058.827} C_VEL
LIN {X 0,Y 728.101,Z 330.529,A -85,B 0,C 180,E1 -1061.364,E2 -1061.364} C_VEL
LIN {X 0,Y 728.137,Z 330.523,A -85,B 0,C 180,E1 -1064.386,E2 -1064.386} C_VEL
LIN {X 0,Y 728.088,Z 330.529,A -85,B 0,C 180,E1 -1066.984,E2 -1066.984} C_VEL
LIN {X 0,Y 728.106,Z 330.528,A -85,B 0,C 180,E1 -1069.556,E2 -1069.556} C_VEL
LIN {X 0,Y 728.128,Z 330.524,A -85,B 0,C 180,E1 -1072.583,E2 -1072.583} C_VEL
LIN {X 0,Y 728.086,Z 330.528,A -85,B 0,C 180,E1 -1075.195,E2 -1075.195} C_VEL
LIN {X 0,Y 728.116,Z 330.531,A -85,B 0,C 180,E1 -1077.796,E2 -1077.796} C_VEL
LIN {X 0,Y 728.111,Z 330.527,A -85,B 0,C 180,E1 -1080.866,E2 -1080.866} C_VEL
LIN {X 0,Y 728.086,Z 330.526,A -85,B 0,C 180,E1 -1083.464,E2 -1083.464} C_VEL
LIN {X 0,Y 728.155,Z 330.533,A -85,B 0,C 180,E1 -1086.228,E2 -1086.228} C_VEL
LIN {X 0,Y 728.096,Z 330.527,A -85,B 0,C 180,E1 -1089.166,E2 -1089.166} C_VEL
LIN {X 0,Y 728.09,Z 330.529,A -85,B 0,C 180,E1 -1091.727,E2 -1091.727} C_VEL
LIN {X 0,Y 728.161,Z 330.529,A -85,B 0,C 180,E1 -1094.554,E2 -1094.554} C_VEL
LIN {X 0,Y 728.092,Z 330.527,A -85,B 0,C 180,E1 -1097.361,E2 -1097.361} C_VEL
LIN {X 0,Y 728.088,Z 330.53,A -85,B 0,C 180,E1 -1099.829,E2 -1099.829} C_VEL
LIN {X 0,Y 728.161,Z 330.529,A -85,B 0,C 180,E1 -1102.665,E2 -1102.665} C_VEL
LIN {X 0,Y 728.095,Z 330.527,A -85,B 0,C 180,E1 -1105.458,E2 -1105.458} C_VEL
LIN {X 0,Y 728.088,Z 330.529,A -85,B 0,C 180,E1 -1107.989,E2 -1107.989} C_VEL
LIN {X 0,Y 728.162,Z 330.528,A -85,B 0,C 180,E1 -1110.81,E2 -1110.81} C_VEL
LIN {X 0,Y 728.09,Z 330.528,A -85,B 0,C 180,E1 -1113.672,E2 -1113.672} C_VEL
LIN {X 0,Y 728.093,Z 330.532,A -85,B 0,C 180,E1 -1116.194,E2 -1116.194} C_VEL
LIN {X 0,Y 728.157,Z 330.524,A -85,B 0,C 180,E1 -1119.118,E2 -1119.118} C_VEL
LIN {X 0,Y 728.086,Z 330.527,A -85,B 0,C 180,E1 -1121.898,E2 -1121.898} C_VEL
LIN {X 0,Y 728.102,Z 330.531,A -85,B 0,C 180,E1 -1124.457,E2 -1124.457} C_VEL
LIN {X 0,Y 728.127,Z 330.528,A -85,B 0,C 180,E1 -1127.513,E2 -1127.513} C_VEL
LIN {X 0,Y 728.085,Z 330.533,A -85,B 0,C 180,E1 -1130.147,E2 -1130.147} C_VEL
LIN {X 0,Y 728.094,Z 330.6,A -85,B 0,C 180,E1 -1132.253,E2 -1132.253} C_VEL
LIN {X 0,Y 731.736,Z 340.724,A -85,B 0,C 180,E1 -1133.202,E2 -1133.202} C_VEL
LIN {X 0,Y 731.312,Z 376.071,A -85,B 0,C 180,E1 -1135.672,E2 -1135.672} C_VEL
LIN {X 0,Y 731.483,Z 377.843,A -85,B 0,C 180,E1 -1135.757,E2 -1135.757} C_VEL
LIN {X 0,Y 733.119,Z 385.198,A -85,B 0,C 180,E1 -1135.929,E2 -1135.929} C_VEL
LIN {X 0,Y 732.284,Z 643.755,A -85,B 0,C 180,E1 -1138.835,E2 -1138.835} C_VEL
LIN {X 0,Y 731.89,Z 766.847,A -85,B 0,C 180,E1 -1140.213,E2 -1140.213} C_VEL
LIN {X 0,Y 731.63,Z 792.376,A -85,B 0,C 180,E1 -1140.64,E2 -1140.64} C_VEL
LIN {X 0,Y 731.417,Z 813.901,A -85,B 0,C 180,E1 -1141.135,E2 -1141.135} C_VEL
LIN {X 0,Y 731.153,Z 837.288,A -85,B 0,C 180,E1 -1141.804,E2 -1141.804} C_VEL
LIN {X 0,Y 730.784,Z 860.275,A -85,B 0,C 180,E1 -1142.622,E2 -1142.622} C_VEL
LIN {X 0,Y 730.481,Z 882.075,A -85,B 0,C 180,E1 -1143.535,E2 -1143.535} C_VEL
LIN {X 0,Y 730.058,Z 903.945,A -85,B 0,C 180,E1 -1144.616,E2 -1144.616} C_VEL
LIN {X 0,Y 729.75,Z 924.342,A -85,B 0,C 180,E1 -1145.772,E2 -1145.772} C_VEL
LIN {X 0,Y 729.365,Z 944.442,A -85,B 0,C 180,E1 -1147.087,E2 -1147.087} C_VEL
LIN {X 0,Y 729.087,Z 963.251,A -85,B 0,C 180,E1 -1148.478,E2 -1148.478} C_VEL
LIN {X 0,Y 728.782,Z 980.461,A -85,B 0,C 180,E1 -1149.94,E2 -1149.94} C_VEL
LIN {X 0,Y 728.57,Z 996.962,A -85,B 0,C 180,E1 -1151.517,E2 -1151.517} C_VEL
LIN {X 0,Y 728.357,Z 1011.448,A -85,B 0,C 180,E1 -1153.107,E2 -1153.107} C_VEL
LIN {X 0,Y 728.222,Z 1025.058,A -85,B 0,C 180,E1 -1154.796,E2 -1154.796} C_VEL
LIN {X 0,Y 728.102,Z 1036.794,A -85,B 0,C 180,E1 -1156.499,E2 -1156.499} C_VEL
LIN {X 0,Y 728.013,Z 1046.95,A -85,B 0,C 180,E1 -1158.191,E2 -1158.191} C_VEL
LIN {X 0,Y 727.951,Z 1056.181,A -85,B 0,C 180,E1 -1160.034,E2 -1160.034} C_VEL
LIN {X 0,Y 727.929,Z 1062.815,A -85,B 0,C 180,E1 -1161.628,E2 -1161.628} C_VEL
LIN {X 0,Y 727.905,Z 1069.244,A -85,B 0,C 180,E1 -1163.532,E2 -1163.532} C_VEL
LIN {X 0,Y 727.917,Z 1073.654,A -85,B 0,C 180,E1 -1165.351,E2 -1165.351} C_VEL
LIN {X 0,Y 727.911,Z 1076.572,A -85,B 0,C 180,E1 -1167.087,E2 -1167.087} C_VEL
LIN {X 0,Y 727.905,Z 1078.262,A -85,B 0,C 180,E1 -1169.134,E2 -1169.134} C_VEL
LIN {X 0,Y 727.899,Z 1078.284,A -85,B 0,C 180,E1 -1170.787,E2 -1170.787} C_VEL
LIN {X 0,Y 727.906,Z 1076.796,A -85,B 0,C 180,E1 -1172.756,E2 -1172.756} C_VEL
LIN {X 0,Y 727.913,Z 1073.813,A -85,B 0,C 180,E1 -1174.57,E2 -1174.57} C_VEL
LIN {X 0,Y 727.907,Z 1069.451,A -85,B 0,C 180,E1 -1176.388,E2 -1176.388} C_VEL
LIN {X 0,Y 727.935,Z 1063.119,A -85,B 0,C 180,E1 -1178.292,E2 -1178.292} C_VEL
LIN {X 0,Y 727.947,Z 1056.536,A -85,B 0,C 180,E1 -1179.886,E2 -1179.886} C_VEL
LIN {X 0,Y 728.016,Z 1047.41,A -85,B 0,C 180,E1 -1181.728,E2 -1181.728} C_VEL
LIN {X 0,Y 728.099,Z 1037.315,A -85,B 0,C 180,E1 -1183.42,E2 -1183.42} C_VEL
LIN {X 0,Y 728.214,Z 1025.49,A -85,B 0,C 180,E1 -1185.143,E2 -1185.143} C_VEL
LIN {X 0,Y 728.358,Z 1011.926,A -85,B 0,C 180,E1 -1186.838,E2 -1186.838} C_VEL
LIN {X 0,Y 728.547,Z 997.74,A -85,B 0,C 180,E1 -1188.401,E2 -1188.401} C_VEL
LIN {X 0,Y 728.773,Z 981.391,A -85,B 0,C 180,E1 -1189.976,E2 -1189.976} C_VEL
LIN {X 0,Y 729.064,Z 964.273,A -85,B 0,C 180,E1 -1191.438,E2 -1191.438} C_VEL
LIN {X 0,Y 729.347,Z 945.651,A -85,B 0,C 180,E1 -1192.829,E2 -1192.829} C_VEL
LIN {X 0,Y 729.719,Z 926.428,A -85,B 0,C 180,E1 -1194.1,E2 -1194.1} C_VEL
LIN {X 0,Y 730.042,Z 905.215,A -85,B 0,C 180,E1 -1195.316,E2 -1195.316} C_VEL
LIN {X 0,Y 730.443,Z 884.086,A -85,B 0,C 180,E1 -1196.372,E2 -1196.372} C_VEL
LIN {X 0,Y 730.773,Z 861.6,A -85,B 0,C 180,E1 -1197.326,E2 -1197.326} C_VEL
LIN {X 0,Y 731.068,Z 840.353,A -85,B 0,C 180,E1 -1198.094,E2 -1198.094} C_VEL
LIN {X 0,Y 731.41,Z 815.372,A -85,B 0,C 180,E1 -1198.827,E2 -1198.827} C_VEL
LIN {X 0,Y 731.614,Z 794.547,A -85,B 0,C 180,E1 -1199.314,E2 -1199.314} C_VEL
LIN {X 0,Y 731.883,Z 769.643,A -85,B 0,C 180,E1 -1199.75,E2 -1199.75} C_VEL
LIN {X 0,Y 732.059,Z 720.364,A -85,B 0,C 180,E1 -1200.319,E2 -1200.319} C_VEL
LIN {X 0,Y 732.828,Z 468.99,A -85,B 0,C 180,E1 -1203.12,E2 -1203.12} C_VEL
LIN {X 0,Y 732.922,Z 383.498,A -85,B 0,C 180,E1 -1204.101,E2 -1204.101} C_VEL
LIN {X 0,Y 731.303,Z 376.686,A -85,B 0,C 180,E1 -1204.285,E2 -1204.285} C_VEL
LIN {X 0,Y 731.729,Z 341.211,A -85,B 0,C 180,E1 -1206.764,E2 -1206.764} C_VEL
LIN {X 0,Y 730.55,Z 337.117,A -85,B 0,C 180,E1 -1207.127,E2 -1207.127} C_VEL
LIN {X 0,Y 728.085,Z 330.536,A -85,B 0,C 180,E1 -1207.77,E2 -1207.77} C_VEL
LIN {X 0,Y 728.114,Z 330.531,A -85,B 0,C 180,E1 -1210.345,E2 -1210.345} C_VEL
LIN {X 0,Y 728.113,Z 330.533,A -85,B 0,C 180,E1 -1213.41,E2 -1213.41} C_VEL
LIN {X 0,Y 728.086,Z 330.53,A -85,B 0,C 180,E1 -1216.023,E2 -1216.023} C_VEL
LIN {X 0,Y 728.156,Z 330.525,A -85,B 0,C 180,E1 -1218.808,E2 -1218.808} C_VEL
LIN {X 0,Y 728.095,Z 330.531,A -85,B 0,C 180,E1 -1221.769,E2 -1221.769} C_VEL
LIN {X 0,Y 728.089,Z 330.518,A -85,B 0,C 180,E1 -1224.292,E2 -1224.292} C_VEL
LIN {X 0,Y 728.161,Z 330.528,A -85,B 0,C 180,E1 -1227.152,E2 -1227.152} C_VEL
LIN {X 0,Y 728.095,Z 330.53,A -85,B 0,C 180,E1 -1229.917,E2 -1229.917} C_VEL
LIN {X 0,Y 728.092,Z 330.525,A -85,B 0,C 180,E1 -1232.432,E2 -1232.432} C_VEL
LIN {X 0,Y 728.162,Z 330.53,A -85,B 0,C 180,E1 -1235.327,E2 -1235.327} C_VEL
LIN {X 0,Y 728.092,Z 330.53,A -85,B 0,C 180,E1 -1238.151,E2 -1238.151} C_VEL
LIN {X 0,Y 728.097,Z 330.526,A -85,B 0,C 180,E1 -1240.673,E2 -1240.673} C_VEL
LIN {X 0,Y 728.155,Z 330.53,A -85,B 0,C 180,E1 -1243.65,E2 -1243.65} C_VEL
LIN {X 0,Y 728.091,Z 330.53,A -85,B 0,C 180,E1 -1246.337,E2 -1246.337} C_VEL
LIN {X 0,Y 728.108,Z 330.524,A -85,B 0,C 180,E1 -1248.915,E2 -1248.915} C_VEL
LIN {X 0,Y 728.133,Z 330.529,A -85,B 0,C 180,E1 -1251.948,E2 -1251.948} C_VEL
LIN {X 0,Y 728.09,Z 330.529,A -85,B 0,C 180,E1 -1254.563,E2 -1254.563} C_VEL
LIN {X 0,Y 728.129,Z 330.523,A -85,B 0,C 180,E1 -1257.245,E2 -1257.245} C_VEL
LIN {X 0,Y 728.108,Z 330.53,A -85,B 0,C 180,E1 -1260.315,E2 -1260.315} C_VEL
LIN {X 0,Y 728.093,Z 330.526,A -85,B 0,C 180,E1 -1262.913,E2 -1262.913} C_VEL
LIN {X 0,Y 728.161,Z 330.527,A -85,B 0,C 180,E1 -1265.753,E2 -1265.753} C_VEL
LIN {X 0,Y 728.098,Z 330.53,A -85,B 0,C 180,E1 -1268.609,E2 -1268.609} C_VEL
LIN {X 0,Y 728.099,Z 330.524,A -85,B 0,C 180,E1 -1271.165,E2 -1271.165} C_VEL
LIN {X 0,Y 728.13,Z 330.525,A -85,B 0,C 180,E1 -1273.523,E2 -1273.523} C_VEL
LIN {X 0,Y 727.207,Z 330.652,A -85,B 0,C 180,E1 -1274.129,E2 -1274.129} C_VEL
LIN {X 0,Y 720.685,Z 331.457,A -85,B 0,C 180,E1 -1275.87,E2 -1275.87} C_VEL
LIN {X 0,Y 720.21,Z 331.52,A -85,B 0,C 180,E1 -1276.267,E2 -1276.267} C_VEL
LIN {X 0,Y 720.153,Z 331.517,A -85,B 0,C 180,E1 -1279.043,E2 -1279.043} C_VEL
LIN {X 0,Y 720.206,Z 331.513,A -85,B 0,C 180,E1 -1281.758,E2 -1281.758} C_VEL
LIN {X 0,Y 720.167,Z 331.52,A -85,B 0,C 180,E1 -1284.791,E2 -1284.791} C_VEL
LIN {X 0,Y 720.158,Z 331.515,A -85,B 0,C 180,E1 -1287.36,E2 -1287.36} C_VEL
LIN {X 0,Y 720.222,Z 331.517,A -85,B 0,C 180,E1 -1290.17,E2 -1290.17} C_VEL
LIN {X 0,Y 720.16,Z 331.519,A -85,B 0,C 180,E1 -1293.069,E2 -1293.069} C_VEL
LIN {X 0,Y 720.171,Z 331.515,A -85,B 0,C 180,E1 -1295.687,E2 -1295.687} C_VEL
LIN {X 0,Y 720.204,Z 331.522,A -85,B 0,C 180,E1 -1298.717,E2 -1298.717} C_VEL
LIN {X 0,Y 720.155,Z 331.519,A -85,B 0,C 180,E1 -1301.431,E2 -1301.431} C_VEL
LIN {X 0,Y 720.22,Z 331.515,A -85,B 0,C 180,E1 -1304.245,E2 -1304.245} C_VEL
LIN {X 0,Y 720.17,Z 331.522,A -85,B 0,C 180,E1 -1307.146,E2 -1307.146} C_VEL
LIN {X 0,Y 720.163,Z 331.519,A -85,B 0,C 180,E1 -1309.788,E2 -1309.788} C_VEL
LIN {X 0,Y 720.222,Z 331.513,A -85,B 0,C 180,E1 -1312.749,E2 -1312.749} C_VEL
LIN {X 0,Y 720.197,Z 331.719,A -85,B 0,C 180,E1 -1313.965,E2 -1313.965} C_VEL
LIN {X 0,Y 724.026,Z 343.373,A -85,B 0,C 180,E1 -1315.08,E2 -1315.08} C_VEL
LIN {X 0,Y 724.097,Z 347.948,A -85,B 0,C 180,E1 -1315.404,E2 -1315.404} C_VEL
LIN {X 0,Y 726.436,Z 357.487,A -85,B 0,C 180,E1 -1315.644,E2 -1315.644} C_VEL
LIN {X 0,Y 725.503,Z 596.713,A -85,B 0,C 180,E1 -1318.362,E2 -1318.362} C_VEL
LIN {X 0,Y 724.939,Z 736.803,A -85,B 0,C 180,E1 -1319.942,E2 -1319.942} C_VEL
LIN {X 0,Y 724.626,Z 762.175,A -85,B 0,C 180,E1 -1320.369,E2 -1320.369} C_VEL
LIN {X 0,Y 724.345,Z 783.933,A -85,B 0,C 180,E1 -1320.872,E2 -1320.872} C_VEL
LIN {X 0,Y 723.993,Z 807.995,A -85,B 0,C 180,E1 -1321.57,E2 -1321.57} C_VEL
LIN {X 0,Y 723.549,Z 830.477,A -85,B 0,C 180,E1 -1322.378,E2 -1322.378} C_VEL
LIN {X 0,Y 723.147,Z 853.169,A -85,B 0,C 180,E1 -1323.341,E2 -1323.341} C_VEL
LIN {X 0,Y 722.62,Z 875.135,A -85,B 0,C 180,E1 -1324.446,E2 -1324.446} C_VEL
LIN {X 0,Y 722.205,Z 896.335,A -85,B 0,C 180,E1 -1325.672,E2 -1325.672} C_VEL
LIN {X 0,Y 721.749,Z 915.627,A -85,B 0,C 180,E1 -1326.96,E2 -1326.96} C_VEL
LIN {X 0,Y 721.363,Z 934.752,A -85,B 0,C 180,E1 -1328.407,E2 -1328.407} C_VEL
LIN {X 0,Y 721.004,Z 951.596,A -85,B 0,C 180,E1 -1329.863,E2 -1329.863} C_VEL
LIN {X 0,Y 720.7,Z 968.878,A -85,B 0,C 180,E1 -1331.559,E2 -1331.559} C_VEL
LIN {X 0,Y 720.468,Z 982.96,A -85,B 0,C 180,E1 -1333.139,E2 -1333.139} C_VEL
LIN {X 0,Y 720.261,Z 997.062,A -85,B 0,C 180,E1 -1334.954,E2 -1334.954} C_VEL
LIN {X 0,Y 720.139,Z 1008.07,A -85,B 0,C 180,E1 -1336.593,E2 -1336.593} C_VEL
LIN {X 0,Y 720.044,Z 1018.887,A -85,B 0,C 180,E1 -1338.465,E2 -1338.465} C_VEL
LIN {X 0,Y 719.959,Z 1027.049,A -85,B 0,C 180,E1 -1340.164,E2 -1340.164} C_VEL
LIN {X 0,Y 719.951,Z 1033.86,A -85,B 0,C 180,E1 -1341.856,E2 -1341.856} C_VEL
LIN {X 0,Y 719.925,Z 1040.161,A -85,B 0,C 180,E1 -1343.861,E2 -1343.861} C_VEL
LIN {X 0,Y 719.916,Z 1044.041,A -85,B 0,C 180,E1 -1345.539,E2 -1345.539} C_VEL
LIN {X 0,Y 719.895,Z 1047.054,A -85,B 0,C 180,E1 -1347.453,E2 -1347.453} C_VEL
LIN {X 0,Y 719.896,Z 1048.294,A -85,B 0,C 180,E1 -1349.284,E2 -1349.284} C_VEL
LIN {X 0,Y 719.915,Z 1048.23,A -85,B 0,C 180,E1 -1351.035,E2 -1351.035} C_VEL
LIN {X 0,Y 719.91,Z 1046.523,A -85,B 0,C 180,E1 -1353.025,E2 -1353.025} C_VEL
LIN {X 0,Y 719.914,Z 1043.744,A -85,B 0,C 180,E1 -1354.7,E2 -1354.7} C_VEL
LIN {X 0,Y 719.914,Z 1039.149,A -85,B 0,C 180,E1 -1356.62,E2 -1356.62} C_VEL
LIN {X 0,Y 719.933,Z 1032.985,A -85,B 0,C 180,E1 -1358.466,E2 -1358.466} C_VEL
LIN {X 0,Y 719.975,Z 1026.38,A -85,B 0,C 180,E1 -1360.078,E2 -1360.078} C_VEL
LIN {X 0,Y 720.057,Z 1016.744,A -85,B 0,C 180,E1 -1362.022,E2 -1362.022} C_VEL
LIN {X 0,Y 720.151,Z 1006.561,A -85,B 0,C 180,E1 -1363.735,E2 -1363.735} C_VEL
LIN {X 0,Y 720.32,Z 994.153,A -85,B 0,C 180,E1 -1365.54,E2 -1365.54} C_VEL
LIN {X 0,Y 720.486,Z 980.895,A -85,B 0,C 180,E1 -1367.194,E2 -1367.194} C_VEL
LIN {X 0,Y 720.771,Z 965.788,A -85,B 0,C 180,E1 -1368.858,E2 -1368.858} C_VEL
LIN {X 0,Y 721.043,Z 949.962,A -85,B 0,C 180,E1 -1370.375,E2 -1370.375} C_VEL
LIN {X 0,Y 721.421,Z 932.185,A -85,B 0,C 180,E1 -1371.891,E2 -1371.891} C_VEL
LIN {X 0,Y 721.795,Z 913.866,A -85,B 0,C 180,E1 -1373.254,E2 -1373.254} C_VEL
LIN {X 0,Y 722.257,Z 892.915,A -85,B 0,C 180,E1 -1374.627,E2 -1374.627} C_VEL
LIN {X 0,Y 722.678,Z 873.164,A -85,B 0,C 180,E1 -1375.75,E2 -1375.75} C_VEL
LIN {X 0,Y 723.185,Z 850.253,A -85,B 0,C 180,E1 -1376.88,E2 -1376.88} C_VEL
LIN {X 0,Y 723.564,Z 829.368,A -85,B 0,C 180,E1 -1377.756,E2 -1377.756} C_VEL
LIN {X 0,Y 724.045,Z 805.898,A -85,B 0,C 180,E1 -1378.588,E2 -1378.588} C_VEL
LIN {X 0,Y 724.355,Z 782.707,A -85,B 0,C 180,E1 -1379.25,E2 -1379.25} C_VEL
LIN {X 0,Y 724.707,Z 759.482,A -85,B 0,C 180,E1 -1379.776,E2 -1379.776} C_VEL
LIN {X 0,Y 724.944,Z 735.287,A -85,B 0,C 180,E1 -1380.167,E2 -1380.167} C_VEL
LIN {X 0,Y 725.989,Z 473.034,A -85,B 0,C 180,E1 -1383.124,E2 -1383.124} C_VEL
LIN {X 0,Y 726.237,Z 355.91,A -85,B 0,C 180,E1 -1384.475,E2 -1384.475} C_VEL
LIN {X 0,Y 723.981,Z 347.461,A -85,B 0,C 180,E1 -1384.701,E2 -1384.701} C_VEL
LIN {X 0,Y 723.96,Z 342.652,A -85,B 0,C 180,E1 -1385.068,E2 -1385.068} C_VEL
LIN {X 0,Y 720.157,Z 331.525,A -85,B 0,C 180,E1 -1386.163,E2 -1386.163} C_VEL
LIN {X 0,Y 720.16,Z 331.524,A -85,B 0,C 180,E1 -1388.769,E2 -1388.769} C_VEL
LIN {X 0,Y 720.22,Z 331.517,A -85,B 0,C 180,E1 -1391.682,E2 -1391.682} C_VEL
LIN {X 0,Y 720.149,Z 331.512,A -85,B 0,C 180,E1 -1394.466,E2 -1394.466} C_VEL
LIN {X 0,Y 720.17,Z 331.523,A -85,B 0,C 180,E1 -1397.028,E2 -1397.028} C_VEL
LIN {X 0,Y 720.176,Z 331.515,A -85,B 0,C 180,E1 -1400.155,E2 -1400.155} C_VEL
LIN {X 0,Y 720.148,Z 331.517,A -85,B 0,C 180,E1 -1402.745,E2 -1402.745} C_VEL
LIN {X 0,Y 720.209,Z 331.52,A -85,B 0,C 180,E1 -1405.497,E2 -1405.497} C_VEL
LIN {X 0,Y 720.159,Z 331.515,A -85,B 0,C 180,E1 -1408.484,E2 -1408.484} C_VEL
LIN {X 0,Y 720.152,Z 331.52,A -85,B 0,C 180,E1 -1411.016,E2 -1411.016} C_VEL
LIN {X 0,Y 720.224,Z 331.52,A -85,B 0,C 180,E1 -1413.801,E2 -1413.801} C_VEL
LIN {X 0,Y 720.154,Z 331.515,A -85,B 0,C 180,E1 -1416.69,E2 -1416.69} C_VEL
LIN {X 0,Y 720.157,Z 331.52,A -85,B 0,C 180,E1 -1419.265,E2 -1419.265} C_VEL
LIN {X 0,Y 720.215,Z 331.515,A -85,B 0,C 180,E1 -1422.216,E2 -1422.216} C_VEL
LIN {X 0,Y 720.149,Z 331.514,A -85,B 0,C 180,E1 -1424.951,E2 -1424.951} C_VEL
LIN {X 0,Y 720.165,Z 331.521,A -85,B 0,C 180,E1 -1427.491,E2 -1427.491} C_VEL
LIN {X 0,Y 720.198,Z 331.515,A -85,B 0,C 180,E1 -1430.49,E2 -1430.49} C_VEL
LIN {X 0,Y 720.149,Z 331.516,A -85,B 0,C 180,E1 -1433.142,E2 -1433.142} C_VEL
LIN {X 0,Y 720.181,Z 331.52,A -85,B 0,C 180,E1 -1435.78,E2 -1435.78} C_VEL
LIN {X 0,Y 720.166,Z 331.514,A -85,B 0,C 180,E1 -1438.886,E2 -1438.886} C_VEL
LIN {X 0,Y 720.148,Z 331.519,A -85,B 0,C 180,E1 -1441.439,E2 -1441.439} C_VEL
LIN {X 0,Y 720.216,Z 331.519,A -85,B 0,C 180,E1 -1444.22,E2 -1444.22} C_VEL
LIN {X 0,Y 720.159,Z 331.514,A -85,B 0,C 180,E1 -1447.098,E2 -1447.098} C_VEL
LIN {X 0,Y 720.151,Z 331.519,A -85,B 0,C 180,E1 -1449.669,E2 -1449.669} C_VEL
LIN {X 0,Y 720.223,Z 331.517,A -85,B 0,C 180,E1 -1452.508,E2 -1452.508} C_VEL
LIN {X 0,Y 720.151,Z 331.517,A -85,B 0,C 180,E1 -1455.379,E2 -1455.379} C_VEL
LIN {X 0,Y 720.152,Z 331.518,A -85,B 0,C 180,E1 -1457.869,E2 -1457.869} C_VEL
LIN {X 0,Y 720.222,Z 331.515,A -85,B 0,C 180,E1 -1460.733,E2 -1460.733} C_VEL
LIN {X 0,Y 720.153,Z 331.516,A -85,B 0,C 180,E1 -1463.484,E2 -1463.484} C_VEL
LIN {X 0,Y 720.155,Z 331.519,A -85,B 0,C 180,E1 -1466.024,E2 -1466.024} C_VEL
LIN {X 0,Y 720.22,Z 331.515,A -85,B 0,C 180,E1 -1468.998,E2 -1468.998} C_VEL
LIN {X 0,Y 720.146,Z 331.517,A -85,B 0,C 180,E1 -1471.751,E2 -1471.751} C_VEL
LIN {X 0,Y 720.166,Z 331.521,A -85,B 0,C 180,E1 -1474.312,E2 -1474.312} C_VEL
LIN {X 0,Y 720.186,Z 331.516,A -85,B 0,C 180,E1 -1477.353,E2 -1477.353} C_VEL
LIN {X 0,Y 720.146,Z 331.516,A -85,B 0,C 180,E1 -1480.005,E2 -1480.005} C_VEL
LIN {X 0,Y 720.201,Z 331.52,A -85,B 0,C 180,E1 -1482.74,E2 -1482.74} C_VEL
